LIN {X 0,Y 514.203,Z 355.204,A -85,B 0,C 180,E1 21211.136,E2 21211.136} C_VEL
LIN {X 0,Y 523.053,Z 367.857,A -85,B 0,C 180,E1 21208.99,E2 21208.99} C_VEL
LIN {X 0,Y 532.804,Z 382.486,A -85,B 0,C 180,E1 21206.835,E2 21206.835} C_VEL
LIN {X 0,Y 543.184,Z 399.298,A -85,B 0,C 180,E1 21204.725,E2 21204.725} C_VEL
LIN {X 0,Y 532.021,Z 628.307,A -85,B 0,C 180,E1 21201.248,E2 21201.248} C_VEL
LIN {X 0,Y 527.564,Z 720.114,A -85,B 0,C 180,E1 21199.84,E2 21199.84} C_VEL
LIN {X 0,Y 524.972,Z 748.17,A -85,B 0,C 180,E1 21199.261,E2 21199.261} C_VEL
LIN {X 0,Y 522.324,Z 769.234,A -85,B 0,C 180,E1 21198.682,E2 21198.682} C_VEL
LIN {X 0,Y 519.318,Z 789.292,A -85,B 0,C 180,E1 21198.004,E2 21198.004} C_VEL
LIN {X 0,Y 515.218,Z 813.189,A -85,B 0,C 180,E1 21197.024,E2 21197.024} C_VEL
LIN {X 0,Y 510.576,Z 836.113,A -85,B 0,C 180,E1 21195.868,E2 21195.868} C_VEL
LIN {X 0,Y 506.148,Z 856.028,A -85,B 0,C 180,E1 21194.69,E2 21194.69} C_VEL
LIN {X 0,Y 500.798,Z 878.497,A -85,B 0,C 180,E1 21193.144,E2 21193.144} C_VEL
LIN {X 0,Y 495.189,Z 899.857,A -85,B 0,C 180,E1 21191.398,E2 21191.398} C_VEL
LIN {X 0,Y 490.436,Z 917.27,A -85,B 0,C 180,E1 21189.77,E2 21189.77} C_VEL
LIN {X 0,Y 484.861,Z 937.229,A -85,B 0,C 180,E1 21187.637,E2 21187.637} C_VEL
LIN {X 0,Y 479.642,Z 955.131,A -85,B 0,C 180,E1 21185.402,E2 21185.402} C_VEL
LIN {X 0,Y 475.369,Z 969.999,A -85,B 0,C 180,E1 21183.297,E2 21183.297} C_VEL
LIN {X 0,Y 470.786,Z 986.437,A -85,B 0,C 180,E1 21180.646,E2 21180.646} C_VEL
LIN {X 0,Y 466.894,Z 1000.666,A -85,B 0,C 180,E1 21177.97,E2 21177.97} C_VEL
LIN {X 0,Y 463.87,Z 1012.654,A -85,B 0,C 180,E1 21175.401,E2 21175.401} C_VEL
LIN {X 0,Y 460.826,Z 1026.036,A -85,B 0,C 180,E1 21172.047,E2 21172.047} C_VEL
LIN {X 0,Y 459.016,Z 1035.196,A -85,B 0,C 180,E1 21169.336,E2 21169.336} C_VEL
LIN {X 0,Y 457.668,Z 1043.402,A -85,B 0,C 180,E1 21166.5,E2 21166.5} C_VEL
LIN {X 0,Y 456.674,Z 1051.232,A -85,B 0,C 180,E1 21163.162,E2 21163.162} C_VEL
LIN {X 0,Y 456.221,Z 1056.208,A -85,B 0,C 180,E1 21160.481,E2 21160.481} C_VEL
LIN {X 0,Y 456.026,Z 1059.887,A -85,B 0,C 180,E1 21157.94,E2 21157.94} C_VEL
LIN {X 0,Y 455.923,Z 1062.661,A -85,B 0,C 180,E1 21155.285,E2 21155.285} C_VEL
LIN {X 0,Y 455.906,Z 1064.554,A -85,B 0,C 180,E1 21152.137,E2 21152.137} C_VEL
LIN {X 0,Y 455.907,Z 1064.806,A -85,B 0,C 180,E1 21149.246,E2 21149.246} C_VEL
LIN {X 0,Y 455.911,Z 1063.998,A -85,B 0,C 180,E1 21146.731,E2 21146.731} C_VEL
LIN {X 0,Y 455.927,Z 1062.196,A -85,B 0,C 180,E1 21144.21,E2 21144.21} C_VEL
LIN {X 0,Y 456.039,Z 1059.388,A -85,B 0,C 180,E1 21141.68,E2 21141.68} C_VEL
LIN {X 0,Y 456.344,Z 1054.717,A -85,B 0,C 180,E1 21138.627,E2 21138.627} C_VEL
LIN {X 0,Y 457.032,Z 1048.041,A -85,B 0,C 180,E1 21135.428,E2 21135.428} C_VEL
LIN {X 0,Y 457.983,Z 1041.122,A -85,B 0,C 180,E1 21132.727,E2 21132.727} C_VEL
LIN {X 0,Y 459.607,Z 1031.801,A -85,B 0,C 180,E1 21129.662,E2 21129.662} C_VEL
LIN {X 0,Y 461.885,Z 1020.576,A -85,B 0,C 180,E1 21126.618,E2 21126.618} C_VEL
LIN {X 0,Y 464.343,Z 1009.773,A -85,B 0,C 180,E1 21124.079,E2 21124.079} C_VEL
LIN {X 0,Y 467.932,Z 995.579,A -85,B 0,C 180,E1 21121.176,E2 21121.176} C_VEL
LIN {X 0,Y 471.825,Z 980.703,A -85,B 0,C 180,E1 21118.579,E2 21118.579} C_VEL
LIN {X 0,Y 475.618,Z 966.792,A -85,B 0,C 180,E1 21116.434,E2 21116.434} C_VEL
LIN {X 0,Y 480.739,Z 948.351,A -85,B 0,C 180,E1 21113.942,E2 21113.942} C_VEL
LIN {X 0,Y 485.605,Z 930.371,A -85,B 0,C 180,E1 21111.851,E2 21111.851} C_VEL
LIN {X 0,Y 490.241,Z 913.03,A -85,B 0,C 180,E1 21110.075,E2 21110.075} C_VEL
LIN {X 0,Y 496.23,Z 889.626,A -85,B 0,C 180,E1 21108.013,E2 21108.013} C_VEL
LIN {X 0,Y 500.877,Z 870.253,A -85,B 0,C 180,E1 21106.551,E2 21106.551} C_VEL
LIN {X 0,Y 505.83,Z 848.283,A -85,B 0,C 180,E1 21105.115,E2 21105.115} C_VEL
LIN {X 0,Y 510.392,Z 825.521,A -85,B 0,C 180,E1 21103.869,E2 21103.869} C_VEL
LIN {X 0,Y 514.144,Z 804.539,A -85,B 0,C 180,E1 21102.896,E2 21102.896} C_VEL
LIN {X 0,Y 517.885,Z 780.938,A -85,B 0,C 180,E1 21101.985,E2 21101.985} C_VEL
LIN {X 0,Y 521.183,Z 755.093,A -85,B 0,C 180,E1 21101.206,E2 21101.206} C_VEL
LIN {X 0,Y 523.436,Z 733.002,A -85,B 0,C 180,E1 21100.696,E2 21100.696} C_VEL
LIN {X 0,Y 525.243,Z 706.485,A -85,B 0,C 180,E1 21100.229,E2 21100.229} C_VEL
LIN {X 0,Y 535.513,Z 472.628,A -85,B 0,C 180,E1 21096.713,E2 21096.713} C_VEL
LIN {X 0,Y 538.83,Z 397.459,A -85,B 0,C 180,E1 21095.558,E2 21095.558} C_VEL
LIN {X 0,Y 529.792,Z 382.604,A -85,B 0,C 180,E1 21093.897,E2 21093.897} C_VEL
LIN {X 0,Y 520.675,Z 368.292,A -85,B 0,C 180,E1 21092.105,E2 21092.105} C_VEL
LIN {X 0,Y 510.021,Z 352.551,A -85,B 0,C 180,E1 21089.833,E2 21089.833} C_VEL
LIN {X 0,Y 499.991,Z 338.758,A -85,B 0,C 180,E1 21087.481,E2 21087.481} C_VEL
LIN {X 0,Y 494.424,Z 331.393,A -85,B 0,C 180,E1 21086.063,E2 21086.063} C_VEL
LIN {X 0,Y 490.131,Z 326.165,A -85,B 0,C 180,E1 21084.915,E2 21084.915} C_VEL
LIN {X 0,Y 486.39,Z 321.608,A -85,B 0,C 180,E1 21083.858,E2 21083.858} C_VEL
LIN {X 0,Y 481.772,Z 316.366,A -85,B 0,C 180,E1 21082.483,E2 21082.483} C_VEL
LIN {X 0,Y 480.461,Z 314.61,A -85,B 0,C 180,E1 21082.064,E2 21082.064} C_VEL
LIN {X 0,Y 477.038,Z 311.21,A -85,B 0,C 180,E1 21080.971,E2 21080.971} C_VEL
LIN {X 0,Y 475.539,Z 308.65,A -85,B 0,C 180,E1 21080.429,E2 21080.429} C_VEL
LIN {X 0,Y 472.204,Z 306.004,A -85,B 0,C 180,E1 21079.289,E2 21079.289} C_VEL
LIN {X 0,Y 469.864,Z 302.242,A -85,B 0,C 180,E1 21078.358,E2 21078.358} C_VEL
LIN {X 0,Y 466.516,Z 299.897,A -85,B 0,C 180,E1 21077.076,E2 21077.076} C_VEL
LIN {X 0,Y 464.568,Z 296.605,A -85,B 0,C 180,E1 21076.184,E2 21076.184} C_VEL
LIN {X 0,Y 463.641,Z 295.554,A -85,B 0,C 180,E1 21075.767,E2 21075.767} C_VEL
LIN {X 0,Y 460.216,Z 293.29,A -85,B 0,C 180,E1 21074.212,E2 21074.212} C_VEL
LIN {X 0,Y 458.544,Z 290.48,A -85,B 0,C 180,E1 21073.268,E2 21073.268} C_VEL
LIN {X 0,Y 458.252,Z 289.079,A -85,B 0,C 180,E1 21072.603,E2 21072.603} C_VEL
LIN {X 0,Y 458.192,Z 288.875,A -85,B 0,C 180,E1 21068.913,E2 21068.913} C_VEL
LIN {X 0,Y 458.169,Z 288.888,A -85,B 0,C 180,E1 21065.385,E2 21065.385} C_VEL
LIN {X 0,Y 458.176,Z 288.901,A -85,B 0,C 180,E1 21061.626,E2 21061.626} C_VEL
LIN {X 0,Y 458.207,Z 288.898,A -85,B 0,C 180,E1 21058.066,E2 21058.066} C_VEL
LIN {X 0,Y 458.22,Z 288.88,A -85,B 0,C 180,E1 21054.365,E2 21054.365} C_VEL
LIN {X 0,Y 458.176,Z 288.875,A -85,B 0,C 180,E1 21050.833,E2 21050.833} C_VEL
LIN {X 0,Y 458.167,Z 288.876,A -85,B 0,C 180,E1 21047.266,E2 21047.266} C_VEL
LIN {X 0,Y 458.249,Z 289.067,A -85,B 0,C 180,E1 21044.172,E2 21044.172} C_VEL
LIN {X 0,Y 458.531,Z 290.412,A -85,B 0,C 180,E1 21043.564,E2 21043.564} C_VEL
LIN {X 0,Y 460.199,Z 293.267,A -85,B 0,C 180,E1 21042.617,E2 21042.617} C_VEL
LIN {X 0,Y 464.437,Z 296.312,A -85,B 0,C 180,E1 21040.703,E2 21040.703} C_VEL
LIN {X 0,Y 466.371,Z 299.715,A -85,B 0,C 180,E1 21039.807,E2 21039.807} C_VEL
LIN {X 0,Y 469.38,Z 302.008,A -85,B 0,C 180,E1 21038.637,E2 21038.637} C_VEL
LIN {X 0,Y 470.174,Z 302.632,A -85,B 0,C 180,E1 21038.341,E2 21038.341} C_VEL
LIN {X 0,Y 472.366,Z 306.213,A -85,B 0,C 180,E1 21037.472,E2 21037.472} C_VEL
LIN {X 0,Y 475.79,Z 309.044,A -85,B 0,C 180,E1 21036.302,E2 21036.302} C_VEL
LIN {X 0,Y 478.497,Z 312.895,A -85,B 0,C 180,E1 21035.366,E2 21035.366} C_VEL
LIN {X 0,Y 481.207,Z 315.37,A -85,B 0,C 180,E1 21034.525,E2 21034.525} C_VEL
LIN {X 0,Y 484.441,Z 319.575,A -85,B 0,C 180,E1 21033.524,E2 21033.524} C_VEL
LIN {X 0,Y 486.437,Z 321.649,A -85,B 0,C 180,E1 21032.949,E2 21032.949} C_VEL
LIN {X 0,Y 490.194,Z 326.225,A -85,B 0,C 180,E1 21031.888,E2 21031.888} C_VEL
LIN {X 0,Y 496.779,Z 334.239,A -85,B 0,C 180,E1 21030.155,E2 21030.155} C_VEL
LIN {X 0,Y 501.543,Z 340.256,A -85,B 0,C 180,E1 21028.979,E2 21028.979} C_VEL
LIN {X 0,Y 509.07,Z 349.89,A -85,B 0,C 180,E1 21027.24,E2 21027.24} C_VEL
LIN {X 0,Y 518.285,Z 362.361,A -85,B 0,C 180,E1 21025.27,E2 21025.27} C_VEL
LIN {X 0,Y 529.578,Z 379.496,A -85,B 0,C 180,E1 21023.033,E2 21023.033} C_VEL
LIN {X 0,Y 538.954,Z 394.907,A -85,B 0,C 180,E1 21021.302,E2 21021.302} C_VEL
LIN {X 0,Y 529.781,Z 598.454,A -85,B 0,C 180,E1 21018.226,E2 21018.226} C_VEL
LIN {X 0,Y 524.636,Z 713.049,A -85,B 0,C 180,E1 21016.486,E2 21016.486} C_VEL
LIN {X 0,Y 522.257,Z 740.771,A -85,B 0,C 180,E1 21015.915,E2 21015.915} C_VEL
LIN {X 0,Y 519.645,Z 763.002,A -85,B 0,C 180,E1 21015.295,E2 21015.295} C_VEL
LIN {X 0,Y 516.831,Z 782.979,A -85,B 0,C 180,E1 21014.61,E2 21014.61} C_VEL
LIN {X 0,Y 512.992,Z 806.654,A -85,B 0,C 180,E1 21013.629,E2 21013.629} C_VEL
LIN {X 0,Y 508.642,Z 829.268,A -85,B 0,C 180,E1 21012.481,E2 21012.481} C_VEL
LIN {X 0,Y 504.692,Z 847.952,A -85,B 0,C 180,E1 21011.378,E2 21011.378} C_VEL
LIN {X 0,Y 500.224,Z 867.614,A -85,B 0,C 180,E1 21010.042,E2 21010.042} C_VEL
LIN {X 0,Y 494.587,Z 890.568,A -85,B 0,C 180,E1 21008.216,E2 21008.216} C_VEL
LIN {X 0,Y 489.946,Z 908.319,A -85,B 0,C 180,E1 21006.578,E2 21006.578} C_VEL
LIN {X 0,Y 485.351,Z 925.361,A -85,B 0,C 180,E1 21004.796,E2 21004.796} C_VEL
LIN {X 0,Y 479.796,Z 945.368,A -85,B 0,C 180,E1 21002.383,E2 21002.383} C_VEL
LIN {X 0,Y 475.603,Z 960.328,A -85,B 0,C 180,E1 21000.302,E2 21000.302} C_VEL
LIN {X 0,Y 471.696,Z 974.528,A -85,B 0,C 180,E1 20998.072,E2 20998.072} C_VEL
LIN {X 0,Y 470.388,Z 979.442,A -85,B 0,C 180,E1 20997.234,E2 20997.234} C_VEL
LIN {X 0,Y 468.274,Z 983.858,A -85,B 0,C 180,E1 20996.497,E2 20996.497} C_VEL
LIN {X 0,Y 459.467,Z 995.612,A -85,B 0,C 180,E1 20994.601,E2 20994.601} C_VEL
LIN {X 0,Y 457.85,Z 998.982,A -85,B 0,C 180,E1 20993.913,E2 20993.913} C_VEL
LIN {X 0,Y 454.838,Z 1010.772,A -85,B 0,C 180,E1 20991.132,E2 20991.132} C_VEL
LIN {X 0,Y 452.659,Z 1020.323,A -85,B 0,C 180,E1 20988.547,E2 20988.547} C_VEL
LIN {X 0,Y 450.633,Z 1030.545,A -85,B 0,C 180,E1 20985.31,E2 20985.31} C_VEL
LIN {X 0,Y 449.378,Z 1038.199,A -85,B 0,C 180,E1 20982.334,E2 20982.334} C_VEL
LIN {X 0,Y 448.644,Z 1043.977,A -85,B 0,C 180,E1 20979.622,E2 20979.622} C_VEL
LIN {X 0,Y 448.188,Z 1049.021,A -85,B 0,C 180,E1 20976.662,E2 20976.662} C_VEL
LIN {X 0,Y 447.969,Z 1053.013,A -85,B 0,C 180,E1 20973.327,E2 20973.327} C_VEL
LIN {X 0,Y 447.928,Z 1055.023,A -85,B 0,C 180,E1 20970.639,E2 20970.639} C_VEL
LIN {X 0,Y 447.907,Z 1055.948,A -85,B 0,C 180,E1 20968.081,E2 20968.081} C_VEL
LIN {X 0,Y 447.905,Z 1055.901,A -85,B 0,C 180,E1 20965.519,E2 20965.519} C_VEL
LIN {X 0,Y 447.921,Z 1054.74,A -85,B 0,C 180,E1 20962.69,E2 20962.69} C_VEL
LIN {X 0,Y 448.033,Z 1051.756,A -85,B 0,C 180,E1 20959.325,E2 20959.325} C_VEL
LIN {X 0,Y 448.263,Z 1047.994,A -85,B 0,C 180,E1 20956.542,E2 20956.542} C_VEL
LIN {X 0,Y 448.757,Z 1043.183,A -85,B 0,C 180,E1 20953.808,E2 20953.808} C_VEL
LIN {X 0,Y 449.736,Z 1036.286,A -85,B 0,C 180,E1 20950.654,E2 20950.654} C_VEL
LIN {X 0,Y 451.296,Z 1027.48,A -85,B 0,C 180,E1 20947.462,E2 20947.462} C_VEL
LIN {X 0,Y 453.17,Z 1018.757,A -85,B 0,C 180,E1 20944.775,E2 20944.775} C_VEL
LIN {X 0,Y 456.012,Z 1007.309,A -85,B 0,C 180,E1 20941.731,E2 20941.731} C_VEL
LIN {X 0,Y 459.523,Z 994.09,A -85,B 0,C 180,E1 20938.776,E2 20938.776} C_VEL
LIN {X 0,Y 463.198,Z 981.437,A -85,B 0,C 180,E1 20936.305,E2 20936.305} C_VEL
LIN {X 0,Y 468.021,Z 965.359,A -85,B 0,C 180,E1 20933.564,E2 20933.564} C_VEL
LIN {X 0,Y 472.912,Z 949.158,A -85,B 0,C 180,E1 20931.194,E2 20931.194} C_VEL
LIN {X 0,Y 477.748,Z 933.313,A -85,B 0,C 180,E1 20929.153,E2 20929.153} C_VEL
LIN {X 0,Y 483.979,Z 912.441,A -85,B 0,C 180,E1 20926.827,E2 20926.827} C_VEL
LIN {X 0,Y 489.009,Z 894.83,A -85,B 0,C 180,E1 20925.136,E2 20925.136} C_VEL
LIN {X 0,Y 493.881,Z 877.04,A -85,B 0,C 180,E1 20923.633,E2 20923.633} C_VEL
LIN {X 0,Y 499.693,Z 854.414,A -85,B 0,C 180,E1 20921.981,E2 20921.981} C_VEL
LIN {X 0,Y 504.539,Z 833.5,A -85,B 0,C 180,E1 20920.693,E2 20920.693} C_VEL
LIN {X 0,Y 508.601,Z 814.32,A -85,B 0,C 180,E1 20919.676,E2 20919.676} C_VEL
LIN {X 0,Y 512.859,Z 791.904,A -85,B 0,C 180,E1 20918.664,E2 20918.664} C_VEL
LIN {X 0,Y 516.841,Z 766.821,A -85,B 0,C 180,E1 20917.754,E2 20917.754} C_VEL
LIN {X 0,Y 519.62,Z 745.455,A -85,B 0,C 180,E1 20917.132,E2 20917.132} C_VEL
LIN {X 0,Y 522.147,Z 721.367,A -85,B 0,C 180,E1 20916.592,E2 20916.592} C_VEL
LIN {X 0,Y 524.302,Z 685.323,A -85,B 0,C 180,E1 20916.003,E2 20916.003} C_VEL
LIN {X 0,Y 535.535,Z 458.38,A -85,B 0,C 180,E1 20912.543,E2 20912.543} C_VEL
LIN {X 0,Y 538.44,Z 400.484,A -85,B 0,C 180,E1 20911.642,E2 20911.642} C_VEL
LIN {X 0,Y 529.82,Z 386.785,A -85,B 0,C 180,E1 20909.852,E2 20909.852} C_VEL
LIN {X 0,Y 520.026,Z 372.01,A -85,B 0,C 180,E1 20907.637,E2 20907.637} C_VEL
LIN {X 0,Y 512.262,Z 361.699,A -85,B 0,C 180,E1 20905.741,E2 20905.741} C_VEL
LIN {X 0,Y 504.417,Z 351.549,A -85,B 0,C 180,E1 20903.635,E2 20903.635} C_VEL
LIN {X 0,Y 499.945,Z 346.055,A -85,B 0,C 180,E1 20902.334,E2 20902.334} C_VEL
LIN {X 0,Y 495.787,Z 340.957,A -85,B 0,C 180,E1 20901.038,E2 20901.038} C_VEL
LIN {X 0,Y 491.944,Z 336.155,A -85,B 0,C 180,E1 20899.75,E2 20899.75} C_VEL
LIN {X 0,Y 487.525,Z 331.174,A -85,B 0,C 180,E1 20898.165,E2 20898.165} C_VEL
LIN {X 0,Y 486.227,Z 329.433,A -85,B 0,C 180,E1 20897.657,E2 20897.657} C_VEL
LIN {X 0,Y 482.681,Z 325.856,A -85,B 0,C 180,E1 20896.24,E2 20896.24} C_VEL
LIN {X 0,Y 480.9,Z 323.244,A -85,B 0,C 180,E1 20895.435,E2 20895.435} C_VEL
LIN {X 0,Y 477.612,Z 320.364,A -85,B 0,C 180,E1 20893.931,E2 20893.931} C_VEL
LIN {X 0,Y 475.685,Z 317.08,A -85,B 0,C 180,E1 20892.874,E2 20892.874} C_VEL
LIN {X 0,Y 471.969,Z 314.314,A -85,B 0,C 180,E1 20890.807,E2 20890.807} C_VEL
LIN {X 0,Y 470.14,Z 311.069,A -85,B 0,C 180,E1 20889.487,E2 20889.487} C_VEL
LIN {X 0,Y 468.4,Z 309.861,A -85,B 0,C 180,E1 20888.223,E2 20888.223} C_VEL
LIN {X 0,Y 465.191,Z 306.945,A -85,B 0,C 180,E1 20885.18,E2 20885.18} C_VEL
LIN {X 0,Y 463.918,Z 304.394,A -85,B 0,C 180,E1 20883.212,E2 20883.212} C_VEL
LIN {X 0,Y 462.586,Z 303.371,A -85,B 0,C 180,E1 20879.628,E2 20879.628} C_VEL
LIN {X 0,Y 463.555,Z 304.007,A -85,B 0,C 180,E1 20874.554,E2 20874.554} C_VEL
LIN {X 0,Y 464.244,Z 304.979,A -85,B 0,C 180,E1 20873.321,E2 20873.321} C_VEL
LIN {X 0,Y 466.922,Z 308.959,A -85,B 0,C 180,E1 20870.084,E2 20870.084} C_VEL
LIN {X 0,Y 470.086,Z 310.878,A -85,B 0,C 180,E1 20867.657,E2 20867.657} C_VEL
LIN {X 0,Y 472,Z 314.284,A -85,B 0,C 180,E1 20866.275,E2 20866.275} C_VEL
LIN {X 0,Y 475.363,Z 316.917,A -85,B 0,C 180,E1 20864.381,E2 20864.381} C_VEL
LIN {X 0,Y 476.013,Z 317.736,A -85,B 0,C 180,E1 20864.028,E2 20864.028} C_VEL
LIN {X 0,Y 478.473,Z 321.384,A -85,B 0,C 180,E1 20862.738,E2 20862.738} C_VEL
LIN {X 0,Y 481.532,Z 323.91,A -85,B 0,C 180,E1 20861.382,E2 20861.382} C_VEL
LIN {X 0,Y 484.662,Z 328.131,A -85,B 0,C 180,E1 20860.035,E2 20860.035} C_VEL
LIN {X 0,Y 486.875,Z 330.162,A -85,B 0,C 180,E1 20859.189,E2 20859.189} C_VEL
LIN {X 0,Y 490.157,Z 334.487,A -85,B 0,C 180,E1 20857.954,E2 20857.954} C_VEL
LIN {X 0,Y 492.165,Z 336.566,A -85,B 0,C 180,E1 20857.262,E2 20857.262} C_VEL
LIN {X 0,Y 496.052,Z 341.208,A -85,B 0,C 180,E1 20855.973,E2 20855.973} C_VEL
LIN {X 0,Y 503.837,Z 351.484,A -85,B 0,C 180,E1 20853.606,E2 20853.606} C_VEL
LIN {X 0,Y 511.816,Z 362.382,A -85,B 0,C 180,E1 20851.435,E2 20851.435} C_VEL
LIN {X 0,Y 520.244,Z 374.603,A -85,B 0,C 180,E1 20849.349,E2 20849.349} C_VEL
LIN {X 0,Y 529.986,Z 389.406,A -85,B 0,C 180,E1 20847.152,E2 20847.152} C_VEL
LIN {X 0,Y 538.508,Z 403.514,A -85,B 0,C 180,E1 20845.37,E2 20845.37} C_VEL
LIN {X 0,Y 526.986,Z 632.03,A -85,B 0,C 180,E1 20841.883,E2 20841.883} C_VEL
LIN {X 0,Y 522.548,Z 720.163,A -85,B 0,C 180,E1 20840.523,E2 20840.523} C_VEL
LIN {X 0,Y 519.868,Z 748.294,A -85,B 0,C 180,E1 20839.94,E2 20839.94} C_VEL
LIN {X 0,Y 517.168,Z 769.128,A -85,B 0,C 180,E1 20839.366,E2 20839.366} C_VEL
LIN {X 0,Y 513.985,Z 789.723,A -85,B 0,C 180,E1 20838.669,E2 20838.669} C_VEL
LIN {X 0,Y 509.53,Z 814.676,A -85,B 0,C 180,E1 20837.632,E2 20837.632} C_VEL
LIN {X 0,Y 504.755,Z 837.376,A -85,B 0,C 180,E1 20836.471,E2 20836.471} C_VEL
LIN {X 0,Y 500.151,Z 857.345,A -85,B 0,C 180,E1 20835.274,E2 20835.274} C_VEL
LIN {X 0,Y 494.381,Z 880.483,A -85,B 0,C 180,E1 20833.648,E2 20833.648} C_VEL
LIN {X 0,Y 489.062,Z 900,A -85,B 0,C 180,E1 20832.034,E2 20832.034} C_VEL
LIN {X 0,Y 484.209,Z 917.111,A -85,B 0,C 180,E1 20830.421,E2 20830.421} C_VEL
LIN {X 0,Y 478.43,Z 937.028,A -85,B 0,C 180,E1 20828.276,E2 20828.276} C_VEL
LIN {X 0,Y 472.943,Z 955.1,A -85,B 0,C 180,E1 20825.997,E2 20825.997} C_VEL
LIN {X 0,Y 468.449,Z 970.051,A -85,B 0,C 180,E1 20823.855,E2 20823.855} C_VEL
LIN {X 0,Y 463.488,Z 986.963,A -85,B 0,C 180,E1 20821.079,E2 20821.079} C_VEL
LIN {X 0,Y 459.565,Z 1000.679,A -85,B 0,C 180,E1 20818.456,E2 20818.456} C_VEL
LIN {X 0,Y 456.368,Z 1012.654,A -85,B 0,C 180,E1 20815.849,E2 20815.849} C_VEL
LIN {X 0,Y 453.258,Z 1025.557,A -85,B 0,C 180,E1 20812.572,E2 20812.572} C_VEL
LIN {X 0,Y 451.312,Z 1034.761,A -85,B 0,C 180,E1 20809.814,E2 20809.814} C_VEL
LIN {X 0,Y 449.91,Z 1042.655,A -85,B 0,C 180,E1 20807.059,E2 20807.059} C_VEL
LIN {X 0,Y 448.796,Z 1050.668,A -85,B 0,C 180,E1 20803.66,E2 20803.66} C_VEL
LIN {X 0,Y 448.271,Z 1055.941,A -85,B 0,C 180,E1 20800.799,E2 20800.799} C_VEL
LIN {X 0,Y 448.036,Z 1059.661,A -85,B 0,C 180,E1 20798.212,E2 20798.212} C_VEL
LIN {X 0,Y 447.924,Z 1062.363,A -85,B 0,C 180,E1 20795.637,E2 20795.637} C_VEL
LIN {X 0,Y 447.913,Z 1064.271,A -85,B 0,C 180,E1 20792.687,E2 20792.687} C_VEL
LIN {X 0,Y 447.903,Z 1064.771,A -85,B 0,C 180,E1 20789.488,E2 20789.488} C_VEL
LIN {X 0,Y 447.912,Z 1063.984,A -85,B 0,C 180,E1 20786.801,E2 20786.801} C_VEL
LIN {X 0,Y 447.932,Z 1062.109,A -85,B 0,C 180,E1 20784.106,E2 20784.106} C_VEL
LIN {X 0,Y 448.048,Z 1059.295,A -85,B 0,C 180,E1 20781.53,E2 20781.53} C_VEL
LIN {X 0,Y 448.378,Z 1054.618,A -85,B 0,C 180,E1 20778.422,E2 20778.422} C_VEL
LIN {X 0,Y 449.108,Z 1047.928,A -85,B 0,C 180,E1 20775.165,E2 20775.165} C_VEL
LIN {X 0,Y 450.068,Z 1041.357,A -85,B 0,C 180,E1 20772.547,E2 20772.547} C_VEL
LIN {X 0,Y 451.615,Z 1032.797,A -85,B 0,C 180,E1 20769.659,E2 20769.659} C_VEL
LIN {X 0,Y 454.14,Z 1020.96,A -85,B 0,C 180,E1 20766.337,E2 20766.337} C_VEL
LIN {X 0,Y 456.71,Z 1010.19,A -85,B 0,C 180,E1 20763.753,E2 20763.753} C_VEL
LIN {X 0,Y 460.33,Z 996.509,A -85,B 0,C 180,E1 20760.886,E2 20760.886} C_VEL
LIN {X 0,Y 464.495,Z 981.283,A -85,B 0,C 180,E1 20758.171,E2 20758.171} C_VEL
LIN {X 0,Y 468.431,Z 967.433,A -85,B 0,C 180,E1 20755.996,E2 20755.996} C_VEL
LIN {X 0,Y 473.547,Z 949.831,A -85,B 0,C 180,E1 20753.56,E2 20753.56} C_VEL
LIN {X 0,Y 478.768,Z 931.23,A -85,B 0,C 180,E1 20751.358,E2 20751.358} C_VEL
LIN {X 0,Y 483.517,Z 914.117,A -85,B 0,C 180,E1 20749.579,E2 20749.579} C_VEL
LIN {X 0,Y 489.181,Z 893.05,A -85,B 0,C 180,E1 20747.667,E2 20747.667} C_VEL
LIN {X 0,Y 494.367,Z 872.191,A -85,B 0,C 180,E1 20746.058,E2 20746.058} C_VEL
LIN {X 0,Y 498.973,Z 852.442,A -85,B 0,C 180,E1 20744.734,E2 20744.734} C_VEL
LIN {X 0,Y 504.099,Z 828.48,A -85,B 0,C 180,E1 20743.368,E2 20743.368} C_VEL
LIN {X 0,Y 508.303,Z 805.834,A -85,B 0,C 180,E1 20742.3,E2 20742.3} C_VEL
LIN {X 0,Y 511.842,Z 784.287,A -85,B 0,C 180,E1 20741.451,E2 20741.451} C_VEL
LIN {X 0,Y 515.633,Z 756.398,A -85,B 0,C 180,E1 20740.582,E2 20740.582} C_VEL
LIN {X 0,Y 518.022,Z 733.825,A -85,B 0,C 180,E1 20740.054,E2 20740.054} C_VEL
LIN {X 0,Y 519.83,Z 708.889,A -85,B 0,C 180,E1 20739.606,E2 20739.606} C_VEL
LIN {X 0,Y 530.5,Z 474.753,A -85,B 0,C 180,E1 20736.063,E2 20736.063} C_VEL
LIN {X 0,Y 533.891,Z 401.34,A -85,B 0,C 180,E1 20734.933,E2 20734.933} C_VEL
LIN {X 0,Y 521.929,Z 381.65,A -85,B 0,C 180,E1 20732.635,E2 20732.635} C_VEL
LIN {X 0,Y 508.905,Z 361.823,A -85,B 0,C 180,E1 20729.873,E2 20729.873} C_VEL
LIN {X 0,Y 498.161,Z 346.708,A -85,B 0,C 180,E1 20727.332,E2 20727.332} C_VEL
LIN {X 0,Y 491.924,Z 338.422,A -85,B 0,C 180,E1 20725.719,E2 20725.719} C_VEL
LIN {X 0,Y 487.786,Z 333.333,A -85,B 0,C 180,E1 20724.59,E2 20724.59} C_VEL
LIN {X 0,Y 483.919,Z 328.472,A -85,B 0,C 180,E1 20723.47,E2 20723.47} C_VEL
LIN {X 0,Y 479.72,Z 323.762,A -85,B 0,C 180,E1 20722.197,E2 20722.197} C_VEL
LIN {X 0,Y 478.423,Z 322.035,A -85,B 0,C 180,E1 20721.776,E2 20721.776} C_VEL
LIN {X 0,Y 474.893,Z 318.339,A -85,B 0,C 180,E1 20720.619,E2 20720.619} C_VEL
LIN {X 0,Y 473.389,Z 316.057,A -85,B 0,C 180,E1 20720.074,E2 20720.074} C_VEL
LIN {X 0,Y 469.99,Z 312.974,A -85,B 0,C 180,E1 20718.867,E2 20718.867} C_VEL
LIN {X 0,Y 467.967,Z 309.826,A -85,B 0,C 180,E1 20718.048,E2 20718.048} C_VEL
LIN {X 0,Y 464.701,Z 307.27,A -85,B 0,C 180,E1 20716.758,E2 20716.758} C_VEL
LIN {X 0,Y 462.413,Z 303.43,A -85,B 0,C 180,E1 20715.682,E2 20715.682} C_VEL
LIN {X 0,Y 458.881,Z 301.098,A -85,B 0,C 180,E1 20714.061,E2 20714.061} C_VEL
LIN {X 0,Y 456.968,Z 298.081,A -85,B 0,C 180,E1 20712.993,E2 20712.993} C_VEL
LIN {X 0,Y 455.974,Z 296.632,A -85,B 0,C 180,E1 20712.41,E2 20712.41} C_VEL
LIN {X 0,Y 452.444,Z 294.447,A -85,B 0,C 180,E1 20710.312,E2 20710.312} C_VEL
LIN {X 0,Y 450.678,Z 291.624,A -85,B 0,C 180,E1 20708.935,E2 20708.935} C_VEL
LIN {X 0,Y 450.328,Z 290.302,A -85,B 0,C 180,E1 20708.17,E2 20708.17} C_VEL
LIN {X 0,Y 450.253,Z 289.888,A -85,B 0,C 180,E1 20705.991,E2 20705.991} C_VEL
LIN {X 0,Y 450.28,Z 289.886,A -85,B 0,C 180,E1 20702.291,E2 20702.291} C_VEL
LIN {X 0,Y 450.254,Z 289.871,A -85,B 0,C 180,E1 20698.727,E2 20698.727} C_VEL
LIN {X 0,Y 450.229,Z 289.864,A -85,B 0,C 180,E1 20695.159,E2 20695.159} C_VEL
LIN {X 0,Y 450.233,Z 289.862,A -85,B 0,C 180,E1 20691.443,E2 20691.443} C_VEL
LIN {X 0,Y 450.298,Z 290.231,A -85,B 0,C 180,E1 20688.732,E2 20688.732} C_VEL
LIN {X 0,Y 450.691,Z 291.628,A -85,B 0,C 180,E1 20687.873,E2 20687.873} C_VEL
LIN {X 0,Y 452.34,Z 294.335,A -85,B 0,C 180,E1 20686.579,E2 20686.579} C_VEL
LIN {X 0,Y 455.62,Z 296.496,A -85,B 0,C 180,E1 20684.601,E2 20684.601} C_VEL
LIN {X 0,Y 456.723,Z 297.434,A -85,B 0,C 180,E1 20683.987,E2 20683.987} C_VEL
LIN {X 0,Y 458.522,Z 300.695,A -85,B 0,C 180,E1 20682.944,E2 20682.944} C_VEL
LIN {X 0,Y 461.991,Z 303.267,A -85,B 0,C 180,E1 20681.318,E2 20681.318} C_VEL
LIN {X 0,Y 462.731,Z 303.898,A -85,B 0,C 180,E1 20680.989,E2 20680.989} C_VEL
LIN {X 0,Y 464.988,Z 307.585,A -85,B 0,C 180,E1 20679.941,E2 20679.941} C_VEL
LIN {X 0,Y 468.353,Z 310.253,A -85,B 0,C 180,E1 20678.621,E2 20678.621} C_VEL
LIN {X 0,Y 470.937,Z 314.109,A -85,B 0,C 180,E1 20677.597,E2 20677.597} C_VEL
LIN {X 0,Y 473.908,Z 316.66,A -85,B 0,C 180,E1 20676.565,E2 20676.565} C_VEL
LIN {X 0,Y 477.043,Z 320.806,A -85,B 0,C 180,E1 20675.48,E2 20675.48} C_VEL
LIN {X 0,Y 479.175,Z 322.836,A -85,B 0,C 180,E1 20674.806,E2 20674.806} C_VEL
LIN {X 0,Y 482.755,Z 327.307,A -85,B 0,C 180,E1 20673.689,E2 20673.689} C_VEL
LIN {X 0,Y 484.432,Z 329.252,A -85,B 0,C 180,E1 20673.192,E2 20673.192} C_VEL
LIN {X 0,Y 488.468,Z 333.963,A -85,B 0,C 180,E1 20672.046,E2 20672.046} C_VEL
LIN {X 0,Y 493.057,Z 339.594,A -85,B 0,C 180,E1 20670.809,E2 20670.809} C_VEL
LIN {X 0,Y 502.322,Z 351.582,A -85,B 0,C 180,E1 20668.499,E2 20668.499} C_VEL
LIN {X 0,Y 513.061,Z 365.837,A -85,B 0,C 180,E1 20666.092,E2 20666.092} C_VEL
LIN {X 0,Y 523.157,Z 381.093,A -85,B 0,C 180,E1 20664.005,E2 20664.005} C_VEL
LIN {X 0,Y 533.472,Z 397.827,A -85,B 0,C 180,E1 20662.03,E2 20662.03} C_VEL
LIN {X 0,Y 533.979,Z 399.099,A -85,B 0,C 180,E1 20661.927,E2 20661.927} C_VEL
LIN {X 0,Y 524.465,Z 602.973,A -85,B 0,C 180,E1 20658.83,E2 20658.83} C_VEL
LIN {X 0,Y 519.337,Z 713.151,A -85,B 0,C 180,E1 20657.146,E2 20657.146} C_VEL
LIN {X 0,Y 516.893,Z 740.867,A -85,B 0,C 180,E1 20656.573,E2 20656.573} C_VEL
LIN {X 0,Y 514.218,Z 762.993,A -85,B 0,C 180,E1 20655.954,E2 20655.954} C_VEL
LIN {X 0,Y 511.414,Z 782.349,A -85,B 0,C 180,E1 20655.291,E2 20655.291} C_VEL
LIN {X 0,Y 507.471,Z 806.004,A -85,B 0,C 180,E1 20654.313,E2 20654.313} C_VEL
LIN {X 0,Y 502.924,Z 829.077,A -85,B 0,C 180,E1 20653.142,E2 20653.142} C_VEL
LIN {X 0,Y 498.65,Z 848.662,A -85,B 0,C 180,E1 20651.978,E2 20651.978} C_VEL
LIN {X 0,Y 493.58,Z 870.279,A -85,B 0,C 180,E1 20650.486,E2 20650.486} C_VEL
LIN {X 0,Y 488.136,Z 891.418,A -85,B 0,C 180,E1 20648.767,E2 20648.767} C_VEL
LIN {X 0,Y 483.448,Z 908.724,A -85,B 0,C 180,E1 20647.151,E2 20647.151} C_VEL
LIN {X 0,Y 478.583,Z 926.121,A -85,B 0,C 180,E1 20645.31,E2 20645.31} C_VEL
LIN {X 0,Y 472.928,Z 945.702,A -85,B 0,C 180,E1 20642.913,E2 20642.913} C_VEL
LIN {X 0,Y 468.562,Z 960.643,A -85,B 0,C 180,E1 20640.807,E2 20640.807} C_VEL
LIN {X 0,Y 464.28,Z 975.584,A -85,B 0,C 180,E1 20638.421,E2 20638.421} C_VEL
LIN {X 0,Y 459.872,Z 991.333,A -85,B 0,C 180,E1 20635.5,E2 20635.5} C_VEL
LIN {X 0,Y 457.85,Z 998.982,A -85,B 0,C 180,E1 20633.913,E2 20633.913} C_VEL
LIN {X 0,Y 455.895,Z 1002.818,A -85,B 0,C 180,E1 20633.101,E2 20633.101} C_VEL
LIN {X 0,Y 447.497,Z 1012.989,A -85,B 0,C 180,E1 20630.986,E2 20630.986} C_VEL
LIN {X 0,Y 446.056,Z 1015.869,A -85,B 0,C 180,E1 20630.239,E2 20630.239} C_VEL
LIN {X 0,Y 443.718,Z 1026.053,A -85,B 0,C 180,E1 20627.164,E2 20627.164} C_VEL
LIN {X 0,Y 442.211,Z 1033.862,A -85,B 0,C 180,E1 20624.402,E2 20624.402} C_VEL
LIN {X 0,Y 441.027,Z 1041.626,A -85,B 0,C 180,E1 20621.111,E2 20621.111} C_VEL
LIN {X 0,Y 440.363,Z 1047.328,A -85,B 0,C 180,E1 20617.961,E2 20617.961} C_VEL
LIN {X 0,Y 440.068,Z 1051.165,A -85,B 0,C 180,E1 20615.214,E2 20615.214} C_VEL
LIN {X 0,Y 439.938,Z 1053.915,A -85,B 0,C 180,E1 20612.475,E2 20612.475} C_VEL
LIN {X 0,Y 439.912,Z 1055.831,A -85,B 0,C 180,E1 20609.219,E2 20609.219} C_VEL
LIN {X 0,Y 439.902,Z 1056.084,A -85,B 0,C 180,E1 20606.09,E2 20606.09} C_VEL
LIN {X 0,Y 439.92,Z 1055.269,A -85,B 0,C 180,E1 20603.475,E2 20603.475} C_VEL
LIN {X 0,Y 439.96,Z 1053.47,A -85,B 0,C 180,E1 20600.846,E2 20600.846} C_VEL
LIN {X 0,Y 440.1,Z 1050.668,A -85,B 0,C 180,E1 20598.201,E2 20598.201} C_VEL
LIN {X 0,Y 440.554,Z 1045.769,A -85,B 0,C 180,E1 20594.87,E2 20594.87} C_VEL
LIN {X 0,Y 441.383,Z 1039.334,A -85,B 0,C 180,E1 20591.657,E2 20591.657} C_VEL
LIN {X 0,Y 442.511,Z 1032.736,A -85,B 0,C 180,E1 20588.941,E2 20588.941} C_VEL
LIN {X 0,Y 444.506,Z 1023.367,A -85,B 0,C 180,E1 20585.692,E2 20585.692} C_VEL
LIN {X 0,Y 447.155,Z 1012.42,A -85,B 0,C 180,E1 20582.572,E2 20582.572} C_VEL
LIN {X 0,Y 449.99,Z 1002.041,A -85,B 0,C 180,E1 20580.003,E2 20580.003} C_VEL
LIN {X 0,Y 454.062,Z 988.309,A -85,B 0,C 180,E1 20577.035,E2 20577.035} C_VEL
LIN {X 0,Y 458.721,Z 973.111,A -85,B 0,C 180,E1 20574.256,E2 20574.256} C_VEL
LIN {X 0,Y 463.195,Z 959.012,A -85,B 0,C 180,E1 20571.992,E2 20571.992} C_VEL
LIN {X 0,Y 469.008,Z 940.795,A -85,B 0,C 180,E1 20569.441,E2 20569.441} C_VEL
LIN {X 0,Y 474.401,Z 923.468,A -85,B 0,C 180,E1 20567.357,E2 20567.357} C_VEL
LIN {X 0,Y 479.653,Z 906.259,A -85,B 0,C 180,E1 20565.539,E2 20565.539} C_VEL
LIN {X 0,Y 486.112,Z 884.161,A -85,B 0,C 180,E1 20563.526,E2 20563.526} C_VEL
LIN {X 0,Y 491.326,Z 864.917,A -85,B 0,C 180,E1 20562.029,E2 20562.029} C_VEL
LIN {X 0,Y 496.383,Z 844.904,A -85,B 0,C 180,E1 20560.677,E2 20560.677} C_VEL
LIN {X 0,Y 502.19,Z 819.535,A -85,B 0,C 180,E1 20559.239,E2 20559.239} C_VEL
LIN {X 0,Y 506.263,Z 799.124,A -85,B 0,C 180,E1 20558.272,E2 20558.272} C_VEL
LIN {X 0,Y 510.03,Z 777.802,A -85,B 0,C 180,E1 20557.427,E2 20557.427} C_VEL
LIN {X 0,Y 514.027,Z 750.288,A -85,B 0,C 180,E1 20556.559,E2 20556.559} C_VEL
LIN {X 0,Y 516.592,Z 727.601,A -85,B 0,C 180,E1 20556.022,E2 20556.022} C_VEL
LIN {X 0,Y 518.508,Z 703.274,A -85,B 0,C 180,E1 20555.581,E2 20555.581} C_VEL
LIN {X 0,Y 530.49,Z 469.255,A -85,B 0,C 180,E1 20551.996,E2 20551.996} C_VEL
LIN {X 0,Y 533.792,Z 404.506,A -85,B 0,C 180,E1 20550.975,E2 20550.975} C_VEL
LIN {X 0,Y 524.258,Z 389.353,A -85,B 0,C 180,E1 20548.914,E2 20548.914} C_VEL
LIN {X 0,Y 516.074,Z 377.179,A -85,B 0,C 180,E1 20546.992,E2 20546.992} C_VEL
LIN {X 0,Y 509.473,Z 368.327,A -85,B 0,C 180,E1 20545.331,E2 20545.331} C_VEL
LIN {X 0,Y 502.035,Z 358.586,A -85,B 0,C 180,E1 20543.288,E2 20543.288} C_VEL
LIN {X 0,Y 497.721,Z 353.216,A -85,B 0,C 180,E1 20542.004,E2 20542.004} C_VEL
LIN {X 0,Y 493.794,Z 348.328,A -85,B 0,C 180,E1 20540.754,E2 20540.754} C_VEL
LIN {X 0,Y 489.856,Z 343.284,A -85,B 0,C 180,E1 20539.403,E2 20539.403} C_VEL
LIN {X 0,Y 485.801,Z 338.743,A -85,B 0,C 180,E1 20537.921,E2 20537.921} C_VEL
LIN {X 0,Y 484.521,Z 337.013,A -85,B 0,C 180,E1 20537.412,E2 20537.412} C_VEL
LIN {X 0,Y 480.905,Z 333.21,A -85,B 0,C 180,E1 20535.929,E2 20535.929} C_VEL
LIN {X 0,Y 479.406,Z 330.959,A -85,B 0,C 180,E1 20535.236,E2 20535.236} C_VEL
LIN {X 0,Y 476.052,Z 327.9,A -85,B 0,C 180,E1 20533.668,E2 20533.668} C_VEL
LIN {X 0,Y 474.26,Z 324.844,A -85,B 0,C 180,E1 20532.666,E2 20532.666} C_VEL
LIN {X 0,Y 470.527,Z 321.89,A -85,B 0,C 180,E1 20530.53,E2 20530.53} C_VEL
LIN {X 0,Y 468.593,Z 318.429,A -85,B 0,C 180,E1 20529.085,E2 20529.085} C_VEL
LIN {X 0,Y 464.516,Z 315.388,A -85,B 0,C 180,E1 20525.559,E2 20525.559} C_VEL
LIN {X 0,Y 462.801,Z 312.206,A -85,B 0,C 180,E1 20522.972,E2 20522.972} C_VEL
LIN {X 0,Y 461.563,Z 311.314,A -85,B 0,C 180,E1 20519.255,E2 20519.255} C_VEL
LIN {X 0,Y 462.646,Z 312.017,A -85,B 0,C 180,E1 20514.419,E2 20514.419} C_VEL
LIN {X 0,Y 463.257,Z 313.073,A -85,B 0,C 180,E1 20513.307,E2 20513.307} C_VEL
LIN {X 0,Y 465.899,Z 316.904,A -85,B 0,C 180,E1 20510.114,E2 20510.114} C_VEL
LIN {X 0,Y 468.78,Z 318.624,A -85,B 0,C 180,E1 20507.872,E2 20507.872} C_VEL
LIN {X 0,Y 470.749,Z 322.091,A -85,B 0,C 180,E1 20506.426,E2 20506.426} C_VEL
LIN {X 0,Y 474.443,Z 325.215,A -85,B 0,C 180,E1 20504.319,E2 20504.319} C_VEL
LIN {X 0,Y 477.026,Z 329.078,A -85,B 0,C 180,E1 20502.935,E2 20502.935} C_VEL
LIN {X 0,Y 479.97,Z 331.623,A -85,B 0,C 180,E1 20501.602,E2 20501.602} C_VEL
LIN {X 0,Y 483.28,Z 335.963,A -85,B 0,C 180,E1 20500.165,E2 20500.165} C_VEL
LIN {X 0,Y 485.239,Z 337.908,A -85,B 0,C 180,E1 20499.399,E2 20499.399} C_VEL
LIN {X 0,Y 488.734,Z 342.339,A -85,B 0,C 180,E1 20498.076,E2 20498.076} C_VEL
LIN {X 0,Y 490.393,Z 344.196,A -85,B 0,C 180,E1 20497.492,E2 20497.492} C_VEL
LIN {X 0,Y 495.406,Z 350.418,A -85,B 0,C 180,E1 20495.813,E2 20495.813} C_VEL
LIN {X 0,Y 501.659,Z 358.782,A -85,B 0,C 180,E1 20493.897,E2 20493.897} C_VEL
LIN {X 0,Y 509.443,Z 369.556,A -85,B 0,C 180,E1 20491.738,E2 20491.738} C_VEL
LIN {X 0,Y 517.559,Z 381.514,A -85,B 0,C 180,E1 20489.687,E2 20489.687} C_VEL
LIN {X 0,Y 527.073,Z 396.154,A -85,B 0,C 180,E1 20487.497,E2 20487.497} C_VEL
LIN {X 0,Y 533.905,Z 407.676,A -85,B 0,C 180,E1 20486.026,E2 20486.026} C_VEL
LIN {X 0,Y 522.054,Z 635.012,A -85,B 0,C 180,E1 20482.542,E2 20482.542} C_VEL
LIN {X 0,Y 517.612,Z 720.189,A -85,B 0,C 180,E1 20481.219,E2 20481.219} C_VEL
LIN {X 0,Y 514.856,Z 748.3,A -85,B 0,C 180,E1 20480.635,E2 20480.635} C_VEL
LIN {X 0,Y 512.067,Z 769.186,A -85,B 0,C 180,E1 20480.06,E2 20480.06} C_VEL
LIN {X 0,Y 508.726,Z 790.162,A -85,B 0,C 180,E1 20479.347,E2 20479.347} C_VEL
LIN {X 0,Y 504.134,Z 814.991,A -85,B 0,C 180,E1 20478.309,E2 20478.309} C_VEL
LIN {X 0,Y 499.217,Z 837.645,A -85,B 0,C 180,E1 20477.144,E2 20477.144} C_VEL
LIN {X 0,Y 494.577,Z 857.135,A -85,B 0,C 180,E1 20475.971,E2 20475.971} C_VEL
LIN {X 0,Y 488.597,Z 880.327,A -85,B 0,C 180,E1 20474.336,E2 20474.336} C_VEL
LIN {X 0,Y 483.079,Z 899.875,A -85,B 0,C 180,E1 20472.71,E2 20472.71} C_VEL
LIN {X 0,Y 477.97,Z 917.237,A -85,B 0,C 180,E1 20471.062,E2 20471.062} C_VEL
LIN {X 0,Y 471.999,Z 937.016,A -85,B 0,C 180,E1 20468.911,E2 20468.911} C_VEL
LIN {X 0,Y 466.265,Z 955.172,A -85,B 0,C 180,E1 20466.595,E2 20466.595} C_VEL
LIN {X 0,Y 461.576,Z 970.107,A -85,B 0,C 180,E1 20464.429,E2 20464.429} C_VEL
LIN {X 0,Y 456.31,Z 987.192,A -85,B 0,C 180,E1 20461.581,E2 20461.581} C_VEL
LIN {X 0,Y 452.269,Z 1000.695,A -85,B 0,C 180,E1 20458.958,E2 20458.958} C_VEL
LIN {X 0,Y 448.896,Z 1012.659,A -85,B 0,C 180,E1 20456.312,E2 20456.312} C_VEL
LIN {X 0,Y 445.614,Z 1025.542,A -85,B 0,C 180,E1 20452.981,E2 20452.981} C_VEL
LIN {X 0,Y 443.551,Z 1034.735,A -85,B 0,C 180,E1 20450.176,E2 20450.176} C_VEL
LIN {X 0,Y 442.046,Z 1042.704,A -85,B 0,C 180,E1 20447.34,E2 20447.34} C_VEL
LIN {X 0,Y 440.831,Z 1050.874,A -85,B 0,C 180,E1 20443.778,E2 20443.778} C_VEL
LIN {X 0,Y 440.282,Z 1056.093,A -85,B 0,C 180,E1 20440.865,E2 20440.865} C_VEL
LIN {X 0,Y 440.037,Z 1059.76,A -85,B 0,C 180,E1 20438.23,E2 20438.23} C_VEL
LIN {X 0,Y 439.923,Z 1062.574,A -85,B 0,C 180,E1 20435.422,E2 20435.422} C_VEL
LIN {X 0,Y 439.907,Z 1064.425,A -85,B 0,C 180,E1 20432.084,E2 20432.084} C_VEL
LIN {X 0,Y 439.908,Z 1064.646,A -85,B 0,C 180,E1 20429.219,E2 20429.219} C_VEL
LIN {X 0,Y 439.911,Z 1063.831,A -85,B 0,C 180,E1 20426.612,E2 20426.612} C_VEL
LIN {X 0,Y 439.937,Z 1062.019,A -85,B 0,C 180,E1 20423.999,E2 20423.999} C_VEL
LIN {X 0,Y 440.055,Z 1059.2,A -85,B 0,C 180,E1 20421.375,E2 20421.375} C_VEL
LIN {X 0,Y 440.415,Z 1054.516,A -85,B 0,C 180,E1 20418.21,E2 20418.21} C_VEL
LIN {X 0,Y 441.153,Z 1048.118,A -85,B 0,C 180,E1 20415.026,E2 20415.026} C_VEL
LIN {X 0,Y 442.215,Z 1041.232,A -85,B 0,C 180,E1 20412.227,E2 20412.227} C_VEL
LIN {X 0,Y 443.77,Z 1033.072,A -85,B 0,C 180,E1 20409.421,E2 20409.421} C_VEL
LIN {X 0,Y 446.401,Z 1021.349,A -85,B 0,C 180,E1 20406.047,E2 20406.047} C_VEL
LIN {X 0,Y 449.094,Z 1010.604,A -85,B 0,C 180,E1 20403.416,E2 20403.416} C_VEL
LIN {X 0,Y 452.481,Z 998.257,A -85,B 0,C 180,E1 20400.767,E2 20400.767} C_VEL
LIN {X 0,Y 457.189,Z 981.859,A -85,B 0,C 180,E1 20397.749,E2 20397.749} C_VEL
LIN {X 0,Y 461.271,Z 968.07,A -85,B 0,C 180,E1 20395.545,E2 20395.545} C_VEL
LIN {X 0,Y 466.035,Z 952.236,A -85,B 0,C 180,E1 20393.307,E2 20393.307} C_VEL
LIN {X 0,Y 471.968,Z 932.086,A -85,B 0,C 180,E1 20390.852,E2 20390.852} C_VEL
LIN {X 0,Y 476.851,Z 915.123,A -85,B 0,C 180,E1 20389.06,E2 20389.06} C_VEL
LIN {X 0,Y 482.532,Z 894.819,A -85,B 0,C 180,E1 20387.182,E2 20387.182} C_VEL
LIN {X 0,Y 488.219,Z 872.812,A -85,B 0,C 180,E1 20385.457,E2 20385.457} C_VEL
LIN {X 0,Y 492.789,Z 853.87,A -85,B 0,C 180,E1 20384.171,E2 20384.171} C_VEL
LIN {X 0,Y 497.838,Z 831.322,A -85,B 0,C 180,E1 20382.854,E2 20382.854} C_VEL
LIN {X 0,Y 502.378,Z 807.902,A -85,B 0,C 180,E1 20381.724,E2 20381.724} C_VEL
LIN {X 0,Y 506.04,Z 786.474,A -85,B 0,C 180,E1 20380.863,E2 20380.863} C_VEL
LIN {X 0,Y 509.731,Z 761.345,A -85,B 0,C 180,E1 20380.042,E2 20380.042} C_VEL
LIN {X 0,Y 512.583,Z 735.621,A -85,B 0,C 180,E1 20379.419,E2 20379.419} C_VEL
LIN {X 0,Y 514.344,Z 713.125,A -85,B 0,C 180,E1 20379.003,E2 20379.003} C_VEL
LIN {X 0,Y 525.425,Z 479.628,A -85,B 0,C 180,E1 20375.443,E2 20375.443} C_VEL
LIN {X 0,Y 528.944,Z 405.214,A -85,B 0,C 180,E1 20374.286,E2 20374.286} C_VEL
LIN {X 0,Y 517.085,Z 385.59,A -85,B 0,C 180,E1 20371.929,E2 20371.929} C_VEL
LIN {X 0,Y 505.105,Z 367.289,A -85,B 0,C 180,E1 20369.305,E2 20369.305} C_VEL
LIN {X 0,Y 495.188,Z 353.177,A -85,B 0,C 180,E1 20366.892,E2 20366.892} C_VEL
LIN {X 0,Y 489.543,Z 345.558,A -85,B 0,C 180,E1 20365.399,E2 20365.399} C_VEL
LIN {X 0,Y 485.261,Z 340.3,A -85,B 0,C 180,E1 20364.208,E2 20364.208} C_VEL
LIN {X 0,Y 480.803,Z 334.835,A -85,B 0,C 180,E1 20362.886,E2 20362.886} C_VEL
LIN {X 0,Y 477.01,Z 330.098,A -85,B 0,C 180,E1 20361.682,E2 20361.682} C_VEL
LIN {X 0,Y 472.765,Z 325.468,A -85,B 0,C 180,E1 20360.263,E2 20360.263} C_VEL
LIN {X 0,Y 471.263,Z 323.416,A -85,B 0,C 180,E1 20359.716,E2 20359.716} C_VEL
LIN {X 0,Y 467.804,Z 319.914,A -85,B 0,C 180,E1 20358.442,E2 20358.442} C_VEL
LIN {X 0,Y 466.088,Z 317.377,A -85,B 0,C 180,E1 20357.736,E2 20357.736} C_VEL
LIN {X 0,Y 462.768,Z 314.463,A -85,B 0,C 180,E1 20356.378,E2 20356.378} C_VEL
LIN {X 0,Y 460.907,Z 311.193,A -85,B 0,C 180,E1 20355.476,E2 20355.476} C_VEL
LIN {X 0,Y 457.314,Z 308.653,A -85,B 0,C 180,E1 20353.788,E2 20353.788} C_VEL
LIN {X 0,Y 455.295,Z 305.326,A -85,B 0,C 180,E1 20352.622,E2 20352.622} C_VEL
LIN {X 0,Y 454.561,Z 304.424,A -85,B 0,C 180,E1 20352.191,E2 20352.191} C_VEL
LIN {X 0,Y 451.105,Z 302.148,A -85,B 0,C 180,E1 20350.085,E2 20350.085} C_VEL
LIN {X 0,Y 449.291,Z 299.156,A -85,B 0,C 180,E1 20348.64,E2 20348.64} C_VEL
LIN {X 0,Y 448.346,Z 297.845,A -85,B 0,C 180,E1 20347.819,E2 20347.819} C_VEL
LIN {X 0,Y 443.018,Z 293.306,A -85,B 0,C 180,E1 20339.741,E2 20339.741} C_VEL
LIN {X 0,Y 442.973,Z 293.254,A -85,B 0,C 180,E1 20337.413,E2 20337.413} C_VEL
LIN {X 0,Y 443.99,Z 294.828,A -85,B 0,C 180,E1 20334.054,E2 20334.054} C_VEL
LIN {X 0,Y 448.895,Z 298.335,A -85,B 0,C 180,E1 20328.542,E2 20328.542} C_VEL
LIN {X 0,Y 450.837,Z 301.85,A -85,B 0,C 180,E1 20326.925,E2 20326.925} C_VEL
LIN {X 0,Y 454.224,Z 304.298,A -85,B 0,C 180,E1 20324.814,E2 20324.814} C_VEL
LIN {X 0,Y 455.159,Z 304.96,A -85,B 0,C 180,E1 20324.291,E2 20324.291} C_VEL
LIN {X 0,Y 457.089,Z 308.391,A -85,B 0,C 180,E1 20323.151,E2 20323.151} C_VEL
LIN {X 0,Y 460.781,Z 311.148,A -85,B 0,C 180,E1 20321.398,E2 20321.398} C_VEL
LIN {X 0,Y 463.61,Z 315.438,A -85,B 0,C 180,E1 20320.076,E2 20320.076} C_VEL
LIN {X 0,Y 466.631,Z 317.972,A -85,B 0,C 180,E1 20318.867,E2 20318.867} C_VEL
LIN {X 0,Y 469.513,Z 321.979,A -85,B 0,C 180,E1 20317.724,E2 20317.724} C_VEL
LIN {X 0,Y 472.101,Z 324.332,A -85,B 0,C 180,E1 20316.807,E2 20316.807} C_VEL
LIN {X 0,Y 475.407,Z 328.523,A -85,B 0,C 180,E1 20315.655,E2 20315.655} C_VEL
LIN {X 0,Y 477.242,Z 330.412,A -85,B 0,C 180,E1 20315.061,E2 20315.061} C_VEL
LIN {X 0,Y 481.074,Z 335.032,A -85,B 0,C 180,E1 20313.856,E2 20313.856} C_VEL
LIN {X 0,Y 487.481,Z 343.055,A -85,B 0,C 180,E1 20311.984,E2 20311.984} C_VEL
LIN {X 0,Y 492.383,Z 349.118,A -85,B 0,C 180,E1 20310.665,E2 20310.665} C_VEL
LIN {X 0,Y 499.519,Z 358.324,A -85,B 0,C 180,E1 20308.873,E2 20308.873} C_VEL
LIN {X 0,Y 510.349,Z 372.932,A -85,B 0,C 180,E1 20306.394,E2 20306.394} C_VEL
LIN {X 0,Y 520.461,Z 388.47,A -85,B 0,C 180,E1 20304.265,E2 20304.265} C_VEL
LIN {X 0,Y 529.094,Z 402.631,A -85,B 0,C 180,E1 20302.575,E2 20302.575} C_VEL
LIN {X 0,Y 519.311,Z 605.301,A -85,B 0,C 180,E1 20299.479,E2 20299.479} C_VEL
LIN {X 0,Y 514.1,Z 713.342,A -85,B 0,C 180,E1 20297.818,E2 20297.818} C_VEL
LIN {X 0,Y 511.534,Z 741.469,A -85,B 0,C 180,E1 20297.231,E2 20297.231} C_VEL
LIN {X 0,Y 508.831,Z 763.189,A -85,B 0,C 180,E1 20296.621,E2 20296.621} C_VEL
LIN {X 0,Y 505.845,Z 783.17,A -85,B 0,C 180,E1 20295.932,E2 20295.932} C_VEL
LIN {X 0,Y 501.79,Z 806.727,A -85,B 0,C 180,E1 20294.95,E2 20294.95} C_VEL
LIN {X 0,Y 497.083,Z 829.766,A -85,B 0,C 180,E1 20293.769,E2 20293.769} C_VEL
LIN {X 0,Y 492.666,Z 849.367,A -85,B 0,C 180,E1 20292.593,E2 20292.593} C_VEL
LIN {X 0,Y 487.284,Z 871.574,A -85,B 0,C 180,E1 20291.043,E2 20291.043} C_VEL
LIN {X 0,Y 481.599,Z 892.746,A -85,B 0,C 180,E1 20289.289,E2 20289.289} C_VEL
LIN {X 0,Y 476.663,Z 910.324,A -85,B 0,C 180,E1 20287.62,E2 20287.62} C_VEL
LIN {X 0,Y 470.943,Z 930.066,A -85,B 0,C 180,E1 20285.473,E2 20285.473} C_VEL
LIN {X 0,Y 465.527,Z 947.857,A -85,B 0,C 180,E1 20283.209,E2 20283.209} C_VEL
LIN {X 0,Y 461.009,Z 962.784,A -85,B 0,C 180,E1 20281.049,E2 20281.049} C_VEL
LIN {X 0,Y 456.035,Z 979.507,A -85,B 0,C 180,E1 20278.268,E2 20278.268} C_VEL
LIN {X 0,Y 452.129,Z 992.843,A -85,B 0,C 180,E1 20275.687,E2 20275.687} C_VEL
LIN {X 0,Y 448.867,Z 1004.686,A -85,B 0,C 180,E1 20273.074,E2 20273.074} C_VEL
LIN {X 0,Y 446.056,Z 1015.869,A -85,B 0,C 180,E1 20270.239,E2 20270.239} C_VEL
LIN {X 0,Y 444.302,Z 1019.142,A -85,B 0,C 180,E1 20269.358,E2 20269.358} C_VEL
LIN {X 0,Y 436.396,Z 1027.534,A -85,B 0,C 180,E1 20267.033,E2 20267.033} C_VEL
LIN {X 0,Y 435.173,Z 1029.952,A -85,B 0,C 180,E1 20266.234,E2 20266.234} C_VEL
LIN {X 0,Y 433.617,Z 1038.24,A -85,B 0,C 180,E1 20262.925,E2 20262.925} C_VEL
LIN {X 0,Y 432.788,Z 1043.885,A -85,B 0,C 180,E1 20260.194,E2 20260.194} C_VEL
LIN {X 0,Y 432.281,Z 1048.489,A -85,B 0,C 180,E1 20257.442,E2 20257.442} C_VEL
LIN {X 0,Y 432.008,Z 1052.679,A -85,B 0,C 180,E1 20254.114,E2 20254.114} C_VEL
LIN {X 0,Y 431.928,Z 1055.087,A -85,B 0,C 180,E1 20250.928,E2 20250.928} C_VEL
LIN {X 0,Y 431.904,Z 1056.073,A -85,B 0,C 180,E1 20248.275,E2 20248.275} C_VEL
LIN {X 0,Y 431.906,Z 1056.087,A -85,B 0,C 180,E1 20245.618,E2 20245.618} C_VEL
LIN {X 0,Y 431.934,Z 1055.124,A -85,B 0,C 180,E1 20242.953,E2 20242.953} C_VEL
LIN {X 0,Y 432.024,Z 1052.624,A -85,B 0,C 180,E1 20239.622,E2 20239.622} C_VEL
LIN {X 0,Y 432.32,Z 1048.37,A -85,B 0,C 180,E1 20236.264,E2 20236.264} C_VEL
LIN {X 0,Y 432.864,Z 1043.677,A -85,B 0,C 180,E1 20233.462,E2 20233.462} C_VEL
LIN {X 0,Y 433.786,Z 1037.781,A -85,B 0,C 180,E1 20230.614,E2 20230.614} C_VEL
LIN {X 0,Y 435.642,Z 1028.472,A -85,B 0,C 180,E1 20226.982,E2 20226.982} C_VEL
LIN {X 0,Y 437.75,Z 1019.639,A -85,B 0,C 180,E1 20224.134,E2 20224.134} C_VEL
LIN {X 0,Y 440.431,Z 1009.763,A -85,B 0,C 180,E1 20221.379,E2 20221.379} C_VEL
LIN {X 0,Y 444.717,Z 995.32,A -85,B 0,C 180,E1 20217.953,E2 20217.953} C_VEL
LIN {X 0,Y 448.75,Z 982.615,A -85,B 0,C 180,E1 20215.377,E2 20215.377} C_VEL
LIN {X 0,Y 453.718,Z 967.537,A -85,B 0,C 180,E1 20212.697,E2 20212.697} C_VEL
LIN {X 0,Y 459.461,Z 950.119,A -85,B 0,C 180,E1 20210.06,E2 20210.06} C_VEL
LIN {X 0,Y 464.391,Z 935.205,A -85,B 0,C 180,E1 20208.084,E2 20208.084} C_VEL
LIN {X 0,Y 470.452,Z 916.638,A -85,B 0,C 180,E1 20205.921,E2 20205.921} C_VEL
LIN {X 0,Y 476.703,Z 896.303,A -85,B 0,C 180,E1 20203.905,E2 20203.905} C_VEL
LIN {X 0,Y 481.898,Z 878.651,A -85,B 0,C 180,E1 20202.383,E2 20202.383} C_VEL
LIN {X 0,Y 487.492,Z 858.499,A -85,B 0,C 180,E1 20200.867,E2 20200.867} C_VEL
LIN {X 0,Y 493.417,Z 834.827,A -85,B 0,C 180,E1 20199.367,E2 20199.367} C_VEL
LIN {X 0,Y 497.768,Z 815.605,A -85,B 0,C 180,E1 20198.334,E2 20198.334} C_VEL
LIN {X 0,Y 501.801,Z 795.669,A -85,B 0,C 180,E1 20197.414,E2 20197.414} C_VEL
LIN {X 0,Y 506.37,Z 769.501,A -85,B 0,C 180,E1 20196.429,E2 20196.429} C_VEL
LIN {X 0,Y 509.524,Z 746.853,A -85,B 0,C 180,E1 20195.759,E2 20195.759} C_VEL
LIN {X 0,Y 512.05,Z 724.325,A -85,B 0,C 180,E1 20195.242,E2 20195.242} C_VEL
LIN {X 0,Y 514.392,Z 690.144,A -85,B 0,C 180,E1 20194.663,E2 20194.663} C_VEL
LIN {X 0,Y 526.453,Z 462.214,A -85,B 0,C 180,E1 20191.158,E2 20191.158} C_VEL
LIN {X 0,Y 529.323,Z 408.799,A -85,B 0,C 180,E1 20190.321,E2 20190.321} C_VEL
LIN {X 0,Y 519.36,Z 392.87,A -85,B 0,C 180,E1 20188.081,E2 20188.081} C_VEL
LIN {X 0,Y 511.186,Z 380.851,A -85,B 0,C 180,E1 20186.08,E2 20186.08} C_VEL
LIN {X 0,Y 502.515,Z 369.404,A -85,B 0,C 180,E1 20183.762,E2 20183.762} C_VEL
LIN {X 0,Y 496.397,Z 361.322,A -85,B 0,C 180,E1 20181.941,E2 20181.941} C_VEL
LIN {X 0,Y 491.479,Z 355.352,A -85,B 0,C 180,E1 20180.359,E2 20180.359} C_VEL
LIN {X 0,Y 487.218,Z 350.018,A -85,B 0,C 180,E1 20178.858,E2 20178.858} C_VEL
LIN {X 0,Y 483.397,Z 345.214,A -85,B 0,C 180,E1 20177.391,E2 20177.391} C_VEL
LIN {X 0,Y 479.018,Z 340.375,A -85,B 0,C 180,E1 20175.559,E2 20175.559} C_VEL
LIN {X 0,Y 477.653,Z 338.499,A -85,B 0,C 180,E1 20174.921,E2 20174.921} C_VEL
LIN {X 0,Y 474.282,Z 335.126,A -85,B 0,C 180,E1 20173.285,E2 20173.285} C_VEL
LIN {X 0,Y 472.617,Z 332.476,A -85,B 0,C 180,E1 20172.338,E2 20172.338} C_VEL
LIN {X 0,Y 469.009,Z 329.341,A -85,B 0,C 180,E1 20170.192,E2 20170.192} C_VEL
LIN {X 0,Y 467.284,Z 326.221,A -85,B 0,C 180,E1 20168.863,E2 20168.863} C_VEL
LIN {X 0,Y 463.431,Z 323.265,A -85,B 0,C 180,E1 20165.448,E2 20165.448} C_VEL
LIN {X 0,Y 461.757,Z 320.094,A -85,B 0,C 180,E1 20162.855,E2 20162.855} C_VEL
LIN {X 0,Y 460.576,Z 319.256,A -85,B 0,C 180,E1 20159.129,E2 20159.129} C_VEL
LIN {X 0,Y 461.674,Z 319.972,A -85,B 0,C 180,E1 20154.407,E2 20154.407} C_VEL
LIN {X 0,Y 462.202,Z 320.971,A -85,B 0,C 180,E1 20153.416,E2 20153.416} C_VEL
LIN {X 0,Y 464.799,Z 324.785,A -85,B 0,C 180,E1 20150.215,E2 20150.215} C_VEL
LIN {X 0,Y 467.55,Z 326.546,A -85,B 0,C 180,E1 20148.027,E2 20148.027} C_VEL
LIN {X 0,Y 469.686,Z 330.107,A -85,B 0,C 180,E1 20146.457,E2 20146.457} C_VEL
LIN {X 0,Y 473.031,Z 333.001,A -85,B 0,C 180,E1 20144.522,E2 20144.522} C_VEL
LIN {X 0,Y 475.704,Z 336.894,A -85,B 0,C 180,E1 20143.075,E2 20143.075} C_VEL
LIN {X 0,Y 478.417,Z 339.315,A -85,B 0,C 180,E1 20141.824,E2 20141.824} C_VEL
LIN {X 0,Y 481.901,Z 343.792,A -85,B 0,C 180,E1 20140.295,E2 20140.295} C_VEL
LIN {X 0,Y 483.544,Z 345.518,A -85,B 0,C 180,E1 20139.64,E2 20139.64} C_VEL
LIN {X 0,Y 487.314,Z 350.183,A -85,B 0,C 180,E1 20138.199,E2 20138.199} C_VEL
LIN {X 0,Y 493.419,Z 357.802,A -85,B 0,C 180,E1 20136.091,E2 20136.091} C_VEL
LIN {X 0,Y 499.495,Z 366.076,A -85,B 0,C 180,E1 20134.19,E2 20134.19} C_VEL
LIN {X 0,Y 507.279,Z 377.01,A -85,B 0,C 180,E1 20131.991,E2 20131.991} C_VEL
LIN {X 0,Y 514.995,Z 388.587,A -85,B 0,C 180,E1 20130.003,E2 20130.003} C_VEL
LIN {X 0,Y 524.068,Z 402.734,A -85,B 0,C 180,E1 20127.87,E2 20127.87} C_VEL
LIN {X 0,Y 529.373,Z 411.829,A -85,B 0,C 180,E1 20126.693,E2 20126.693} C_VEL
LIN {X 0,Y 517.2,Z 637.889,A -85,B 0,C 180,E1 20123.215,E2 20123.215} C_VEL
LIN {X 0,Y 512.756,Z 720.179,A -85,B 0,C 180,E1 20121.93,E2 20121.93} C_VEL
LIN {X 0,Y 509.921,Z 748.305,A -85,B 0,C 180,E1 20121.344,E2 20121.344} C_VEL
LIN {X 0,Y 507.068,Z 769.072,A -85,B 0,C 180,E1 20120.773,E2 20120.773} C_VEL
LIN {X 0,Y 503.66,Z 789.87,A -85,B 0,C 180,E1 20120.067,E2 20120.067} C_VEL
LIN {X 0,Y 499.06,Z 814.189,A -85,B 0,C 180,E1 20119.054,E2 20119.054} C_VEL
LIN {X 0,Y 493.986,Z 836.922,A -85,B 0,C 180,E1 20117.888,E2 20117.888} C_VEL
LIN {X 0,Y 489.136,Z 856.721,A -85,B 0,C 180,E1 20116.696,E2 20116.696} C_VEL
LIN {X 0,Y 483.18,Z 879.199,A -85,B 0,C 180,E1 20115.116,E2 20115.116} C_VEL
LIN {X 0,Y 477.205,Z 899.635,A -85,B 0,C 180,E1 20113.413,E2 20113.413} C_VEL
LIN {X 0,Y 471.795,Z 917.366,A -85,B 0,C 180,E1 20111.718,E2 20111.718} C_VEL
LIN {X 0,Y 465.423,Z 937.612,A -85,B 0,C 180,E1 20109.487,E2 20109.487} C_VEL
LIN {X 0,Y 459.639,Z 955.247,A -85,B 0,C 180,E1 20107.211,E2 20107.211} C_VEL
LIN {X 0,Y 454.752,Z 970.166,A -85,B 0,C 180,E1 20105.021,E2 20105.021} C_VEL
LIN {X 0,Y 449.239,Z 987.224,A -85,B 0,C 180,E1 20102.137,E2 20102.137} C_VEL
LIN {X 0,Y 445.003,Z 1000.715,A -85,B 0,C 180,E1 20099.477,E2 20099.477} C_VEL
LIN {X 0,Y 441.461,Z 1012.666,A -85,B 0,C 180,E1 20096.79,E2 20096.79} C_VEL
LIN {X 0,Y 437.995,Z 1025.529,A -85,B 0,C 180,E1 20093.404,E2 20093.404} C_VEL
LIN {X 0,Y 435.805,Z 1034.713,A -85,B 0,C 180,E1 20090.551,E2 20090.551} C_VEL
LIN {X 0,Y 434.147,Z 1042.989,A -85,B 0,C 180,E1 20087.542,E2 20087.542} C_VEL
LIN {X 0,Y 432.905,Z 1050.828,A -85,B 0,C 180,E1 20084.035,E2 20084.035} C_VEL
LIN {X 0,Y 432.329,Z 1055.832,A -85,B 0,C 180,E1 20081.202,E2 20081.202} C_VEL
LIN {X 0,Y 432.045,Z 1059.701,A -85,B 0,C 180,E1 20078.384,E2 20078.384} C_VEL
LIN {X 0,Y 431.923,Z 1062.46,A -85,B 0,C 180,E1 20075.58,E2 20075.58} C_VEL
LIN {X 0,Y 431.908,Z 1064.326,A -85,B 0,C 180,E1 20072.256,E2 20072.256} C_VEL
LIN {X 0,Y 431.908,Z 1064.566,A -85,B 0,C 180,E1 20069.204,E2 20069.204} C_VEL
LIN {X 0,Y 431.911,Z 1063.745,A -85,B 0,C 180,E1 20066.549,E2 20066.549} C_VEL
LIN {X 0,Y 431.942,Z 1061.928,A -85,B 0,C 180,E1 20063.887,E2 20063.887} C_VEL
LIN {X 0,Y 432.063,Z 1059.062,A -85,B 0,C 180,E1 20061.181,E2 20061.181} C_VEL
LIN {X 0,Y 432.484,Z 1054.185,A -85,B 0,C 180,E1 20057.855,E2 20057.855} C_VEL
LIN {X 0,Y 433.288,Z 1047.692,A -85,B 0,C 180,E1 20054.61,E2 20054.61} C_VEL
LIN {X 0,Y 434.373,Z 1041.104,A -85,B 0,C 180,E1 20051.895,E2 20051.895} C_VEL
LIN {X 0,Y 436.117,Z 1032.524,A -85,B 0,C 180,E1 20048.903,E2 20048.903} C_VEL
LIN {X 0,Y 438.896,Z 1020.801,A -85,B 0,C 180,E1 20045.504,E2 20045.504} C_VEL
LIN {X 0,Y 441.655,Z 1010.435,A -85,B 0,C 180,E1 20042.932,E2 20042.932} C_VEL
LIN {X 0,Y 445.198,Z 998.075,A -85,B 0,C 180,E1 20040.241,E2 20040.241} C_VEL
LIN {X 0,Y 449.906,Z 982.432,A -85,B 0,C 180,E1 20037.313,E2 20037.313} C_VEL
LIN {X 0,Y 454.432,Z 967.77,A -85,B 0,C 180,E1 20034.937,E2 20034.937} C_VEL
LIN {X 0,Y 459.656,Z 951.089,A -85,B 0,C 180,E1 20032.56,E2 20032.56} C_VEL
LIN {X 0,Y 465.538,Z 931.816,A -85,B 0,C 180,E1 20030.205,E2 20030.205} C_VEL
LIN {X 0,Y 470.553,Z 915.012,A -85,B 0,C 180,E1 20028.416,E2 20028.416} C_VEL
LIN {X 0,Y 476.496,Z 894.508,A -85,B 0,C 180,E1 20026.506,E2 20026.506} C_VEL
LIN {X 0,Y 482.322,Z 872.671,A -85,B 0,C 180,E1 20024.786,E2 20024.786} C_VEL
LIN {X 0,Y 487.099,Z 853.474,A -85,B 0,C 180,E1 20023.478,E2 20023.478} C_VEL
LIN {X 0,Y 492.541,Z 829.815,A -85,B 0,C 180,E1 20022.099,E2 20022.099} C_VEL
LIN {X 0,Y 497.116,Z 806.658,A -85,B 0,C 180,E1 20020.991,E2 20020.991} C_VEL
LIN {X 0,Y 500.709,Z 786.107,A -85,B 0,C 180,E1 20020.167,E2 20020.167} C_VEL
LIN {X 0,Y 504.538,Z 760.57,A -85,B 0,C 180,E1 20019.336,E2 20019.336} C_VEL
LIN {X 0,Y 507.41,Z 735.271,A -85,B 0,C 180,E1 20018.725,E2 20018.725} C_VEL
LIN {X 0,Y 509.216,Z 712.688,A -85,B 0,C 180,E1 20018.308,E2 20018.308} C_VEL
LIN {X 0,Y 520.668,Z 479.327,A -85,B 0,C 180,E1 20014.731,E2 20014.731} C_VEL
LIN {X 0,Y 524.153,Z 409.159,A -85,B 0,C 180,E1 20013.642,E2 20013.642} C_VEL
LIN {X 0,Y 513.24,Z 391.067,A -85,B 0,C 180,E1 20011.409,E2 20011.409} C_VEL
LIN {X 0,Y 501.901,Z 373.521,A -85,B 0,C 180,E1 20008.856,E2 20008.856} C_VEL
LIN {X 0,Y 492.242,Z 359.632,A -85,B 0,C 180,E1 20006.447,E2 20006.447} C_VEL
LIN {X 0,Y 487.079,Z 352.58,A -85,B 0,C 180,E1 20005.049,E2 20005.049} C_VEL
LIN {X 0,Y 482.856,Z 347.352,A -85,B 0,C 180,E1 20003.849,E2 20003.849} C_VEL
LIN {X 0,Y 478.555,Z 342.017,A -85,B 0,C 180,E1 20002.545,E2 20002.545} C_VEL
LIN {X 0,Y 474.038,Z 336.541,A -85,B 0,C 180,E1 20001.078,E2 20001.078} C_VEL
LIN {X 0,Y 470.348,Z 332.113,A -85,B 0,C 180,E1 19999.788,E2 19999.788} C_VEL
LIN {X 0,Y 469.159,Z 330.736,A -85,B 0,C 180,E1 19999.354,E2 19999.354} C_VEL
LIN {X 0,Y 465.716,Z 326.946,A -85,B 0,C 180,E1 19998.041,E2 19998.041} C_VEL
LIN {X 0,Y 464.53,Z 325.082,A -85,B 0,C 180,E1 19997.539,E2 19997.539} C_VEL
LIN {X 0,Y 461.117,Z 321.998,A -85,B 0,C 180,E1 19996.115,E2 19996.115} C_VEL
LIN {X 0,Y 459.136,Z 318.81,A -85,B 0,C 180,E1 19995.149,E2 19995.149} C_VEL
LIN {X 0,Y 455.532,Z 315.933,A -85,B 0,C 180,E1 19993.39,E2 19993.39} C_VEL
LIN {X 0,Y 453.378,Z 312.305,A -85,B 0,C 180,E1 19992.094,E2 19992.094} C_VEL
LIN {X 0,Y 449.95,Z 310.035,A -85,B 0,C 180,E1 19989.982,E2 19989.982} C_VEL
LIN {X 0,Y 448.071,Z 307.029,A -85,B 0,C 180,E1 19988.469,E2 19988.469} C_VEL
LIN {X 0,Y 447.373,Z 305.841,A -85,B 0,C 180,E1 19987.836,E2 19987.836} C_VEL
LIN {X 0,Y 442.023,Z 301.222,A -85,B 0,C 180,E1 19979.611,E2 19979.611} C_VEL
LIN {X 0,Y 442.012,Z 301.228,A -85,B 0,C 180,E1 19977.277,E2 19977.277} C_VEL
LIN {X 0,Y 443.217,Z 303.099,A -85,B 0,C 180,E1 19973.653,E2 19973.653} C_VEL
LIN {X 0,Y 447.746,Z 306.208,A -85,B 0,C 180,E1 19968.666,E2 19968.666} C_VEL
LIN {X 0,Y 449.522,Z 309.554,A -85,B 0,C 180,E1 19967.148,E2 19967.148} C_VEL
LIN {X 0,Y 453.055,Z 312.184,A -85,B 0,C 180,E1 19964.905,E2 19964.905} C_VEL
LIN {X 0,Y 453.747,Z 312.812,A -85,B 0,C 180,E1 19964.503,E2 19964.503} C_VEL
LIN {X 0,Y 455.892,Z 316.352,A -85,B 0,C 180,E1 19963.237,E2 19963.237} C_VEL
LIN {X 0,Y 459.534,Z 319.363,A -85,B 0,C 180,E1 19961.477,E2 19961.477} C_VEL
LIN {X 0,Y 462.205,Z 323.25,A -85,B 0,C 180,E1 19960.225,E2 19960.225} C_VEL
LIN {X 0,Y 464.924,Z 325.64,A -85,B 0,C 180,E1 19959.116,E2 19959.116} C_VEL
LIN {X 0,Y 467.936,Z 329.684,A -85,B 0,C 180,E1 19957.909,E2 19957.909} C_VEL
LIN {X 0,Y 470.264,Z 331.899,A -85,B 0,C 180,E1 19957.068,E2 19957.068} C_VEL
LIN {X 0,Y 473.777,Z 336.233,A -85,B 0,C 180,E1 19955.831,E2 19955.831} C_VEL
LIN {X 0,Y 475.404,Z 338.089,A -85,B 0,C 180,E1 19955.29,E2 19955.29} C_VEL
LIN {X 0,Y 480.28,Z 344.114,A -85,B 0,C 180,E1 19953.743,E2 19953.743} C_VEL
LIN {X 0,Y 485.352,Z 350.475,A -85,B 0,C 180,E1 19952.251,E2 19952.251} C_VEL
LIN {X 0,Y 490.303,Z 356.67,A -85,B 0,C 180,E1 19950.897,E2 19950.897} C_VEL
LIN {X 0,Y 497.689,Z 366.411,A -85,B 0,C 180,E1 19949.014,E2 19949.014} C_VEL
LIN {X 0,Y 507.653,Z 380.018,A -85,B 0,C 180,E1 19946.699,E2 19946.699} C_VEL
LIN {X 0,Y 518.5,Z 396.934,A -85,B 0,C 180,E1 19944.381,E2 19944.381} C_VEL
LIN {X 0,Y 524.247,Z 406.793,A -85,B 0,C 180,E1 19943.224,E2 19943.224} C_VEL
LIN {X 0,Y 514.014,Z 611.922,A -85,B 0,C 180,E1 19940.076,E2 19940.076} C_VEL
LIN {X 0,Y 508.935,Z 713.519,A -85,B 0,C 180,E1 19938.503,E2 19938.503} C_VEL
LIN {X 0,Y 506.292,Z 741.672,A -85,B 0,C 180,E1 19937.914,E2 19937.914} C_VEL
LIN {X 0,Y 503.544,Z 763.161,A -85,B 0,C 180,E1 19937.309,E2 19937.309} C_VEL
LIN {X 0,Y 500.571,Z 782.523,A -85,B 0,C 180,E1 19936.642,E2 19936.642} C_VEL
LIN {X 0,Y 496.368,Z 806.315,A -85,B 0,C 180,E1 19935.652,E2 19935.652} C_VEL
LIN {X 0,Y 491.371,Z 830.148,A -85,B 0,C 180,E1 19934.427,E2 19934.427} C_VEL
LIN {X 0,Y 487.002,Z 848.957,A -85,B 0,C 180,E1 19933.294,E2 19933.294} C_VEL
LIN {X 0,Y 481.618,Z 870.474,A -85,B 0,C 180,E1 19931.792,E2 19931.792} C_VEL
LIN {X 0,Y 475.731,Z 891.856,A -85,B 0,C 180,E1 19930.027,E2 19930.027} C_VEL
LIN {X 0,Y 470.601,Z 909.523,A -85,B 0,C 180,E1 19928.346,E2 19928.346} C_VEL
LIN {X 0,Y 464.863,Z 928.677,A -85,B 0,C 180,E1 19926.264,E2 19926.264} C_VEL
LIN {X 0,Y 459.017,Z 947.272,A -85,B 0,C 180,E1 19923.893,E2 19923.893} C_VEL
LIN {X 0,Y 454.336,Z 962.096,A -85,B 0,C 180,E1 19921.734,E2 19921.734} C_VEL
LIN {X 0,Y 449.278,Z 978.399,A -85,B 0,C 180,E1 19919.023,E2 19919.023} C_VEL
LIN {X 0,Y 444.955,Z 992.474,A -85,B 0,C 180,E1 19916.276,E2 19916.276} C_VEL
LIN {X 0,Y 441.663,Z 1003.764,A -85,B 0,C 180,E1 19913.764,E2 19913.764} C_VEL
LIN {X 0,Y 438.486,Z 1015.776,A -85,B 0,C 180,E1 19910.698,E2 19910.698} C_VEL
LIN {X 0,Y 435.942,Z 1026.234,A -85,B 0,C 180,E1 19907.485,E2 19907.485} C_VEL
LIN {X 0,Y 435.173,Z 1029.952,A -85,B 0,C 180,E1 19906.234,E2 19906.234} C_VEL
LIN {X 0,Y 433.67,Z 1032.661,A -85,B 0,C 180,E1 19905.295,E2 19905.295} C_VEL
LIN {X 0,Y 426.174,Z 1039.363,A -85,B 0,C 180,E1 19902.711,E2 19902.711} C_VEL
LIN {X 0,Y 425.286,Z 1041.117,A -85,B 0,C 180,E1 19901.931,E2 19901.931} C_VEL
LIN {X 0,Y 424.455,Z 1047.2,A -85,B 0,C 180,E1 19898.535,E2 19898.535} C_VEL
LIN {X 0,Y 424.101,Z 1051.101,A -85,B 0,C 180,E1 19895.683,E2 19895.683} C_VEL
LIN {X 0,Y 423.956,Z 1053.802,A -85,B 0,C 180,E1 19892.974,E2 19892.974} C_VEL
LIN {X 0,Y 423.935,Z 1055.657,A -85,B 0,C 180,E1 19890,E2 19890} C_VEL
LIN {X 0,Y 423.9,Z 1056.338,A -85,B 0,C 180,E1 19886.619,E2 19886.619} C_VEL
LIN {X 0,Y 423.921,Z 1055.52,A -85,B 0,C 180,E1 19883.499,E2 19883.499} C_VEL
LIN {X 0,Y 423.967,Z 1053.784,A -85,B 0,C 180,E1 19880.772,E2 19880.772} C_VEL
LIN {X 0,Y 424.122,Z 1051.048,A -85,B 0,C 180,E1 19878.026,E2 19878.026} C_VEL
LIN {X 0,Y 424.554,Z 1046.794,A -85,B 0,C 180,E1 19874.932,E2 19874.932} C_VEL
LIN {X 0,Y 425.518,Z 1040.201,A -85,B 0,C 180,E1 19871.363,E2 19871.363} C_VEL
LIN {X 0,Y 426.816,Z 1033.406,A -85,B 0,C 180,E1 19868.42,E2 19868.42} C_VEL
LIN {X 0,Y 428.705,Z 1025.329,A -85,B 0,C 180,E1 19865.471,E2 19865.471} C_VEL
LIN {X 0,Y 431.957,Z 1013.322,A -85,B 0,C 180,E1 19861.822,E2 19861.822} C_VEL
LIN {X 0,Y 435.26,Z 1002.455,A -85,B 0,C 180,E1 19859.031,E2 19859.031} C_VEL
LIN {X 0,Y 439.717,Z 988.828,A -85,B 0,C 180,E1 19855.987,E2 19855.987} C_VEL
LIN {X 0,Y 444.844,Z 973.623,A -85,B 0,C 180,E1 19853.12,E2 19853.12} C_VEL
LIN {X 0,Y 449.626,Z 959.78,A -85,B 0,C 180,E1 19850.834,E2 19850.834} C_VEL
LIN {X 0,Y 455.667,Z 942.452,A -85,B 0,C 180,E1 19848.327,E2 19848.327} C_VEL
LIN {X 0,Y 461.837,Z 924.099,A -85,B 0,C 180,E1 19846.068,E2 19846.068} C_VEL
LIN {X 0,Y 467.456,Z 907.003,A -85,B 0,C 180,E1 19844.229,E2 19844.229} C_VEL
LIN {X 0,Y 474.151,Z 885.777,A -85,B 0,C 180,E1 19842.253,E2 19842.253} C_VEL
LIN {X 0,Y 479.92,Z 865.875,A -85,B 0,C 180,E1 19840.679,E2 19840.679} C_VEL
LIN {X 0,Y 485.048,Z 846.867,A -85,B 0,C 180,E1 19839.373,E2 19839.373} C_VEL
LIN {X 0,Y 490.95,Z 823.115,A -85,B 0,C 180,E1 19837.985,E2 19837.985} C_VEL
LIN {X 0,Y 495.754,Z 800.575,A -85,B 0,C 180,E1 19836.899,E2 19836.899} C_VEL
LIN {X 0,Y 499.681,Z 779.691,A -85,B 0,C 180,E1 19836.058,E2 19836.058} C_VEL
LIN {X 0,Y 503.755,Z 754.157,A -85,B 0,C 180,E1 19835.225,E2 19835.225} C_VEL
LIN {X 0,Y 506.77,Z 729.199,A -85,B 0,C 180,E1 19834.619,E2 19834.619} C_VEL
LIN {X 0,Y 508.705,Z 706.721,A -85,B 0,C 180,E1 19834.201,E2 19834.201} C_VEL
LIN {X 0,Y 521.545,Z 472.941,A -85,B 0,C 180,E1 19830.586,E2 19830.586} C_VEL
LIN {X 0,Y 524.836,Z 412.971,A -85,B 0,C 180,E1 19829.636,E2 19829.636} C_VEL
LIN {X 0,Y 514.963,Z 397.256,A -85,B 0,C 180,E1 19827.336,E2 19827.336} C_VEL
LIN {X 0,Y 508.277,Z 387.326,A -85,B 0,C 180,E1 19825.645,E2 19825.645} C_VEL
LIN {X 0,Y 498.241,Z 373.703,A -85,B 0,C 180,E1 19822.85,E2 19822.85} C_VEL
LIN {X 0,Y 490.18,Z 363.397,A -85,B 0,C 180,E1 19820.29,E2 19820.29} C_VEL
LIN {X 0,Y 485.164,Z 357.258,A -85,B 0,C 180,E1 19818.505,E2 19818.505} C_VEL
LIN {X 0,Y 480.851,Z 351.916,A -85,B 0,C 180,E1 19816.801,E2 19816.801} C_VEL
LIN {X 0,Y 477.152,Z 347.534,A -85,B 0,C 180,E1 19815.185,E2 19815.185} C_VEL
LIN {X 0,Y 476.175,Z 346.205,A -85,B 0,C 180,E1 19814.719,E2 19814.719} C_VEL
LIN {X 0,Y 472.854,Z 342.818,A -85,B 0,C 180,E1 19813.077,E2 19813.077} C_VEL
LIN {X 0,Y 471.211,Z 340.224,A -85,B 0,C 180,E1 19812.127,E2 19812.127} C_VEL
LIN {X 0,Y 467.594,Z 336.903,A -85,B 0,C 180,E1 19809.912,E2 19809.912} C_VEL
LIN {X 0,Y 465.98,Z 334.026,A -85,B 0,C 180,E1 19808.639,E2 19808.639} C_VEL
LIN {X 0,Y 462.248,Z 330.991,A -85,B 0,C 180,E1 19805.213,E2 19805.213} C_VEL
LIN {X 0,Y 460.714,Z 327.984,A -85,B 0,C 180,E1 19802.737,E2 19802.737} C_VEL
LIN {X 0,Y 459.584,Z 327.199,A -85,B 0,C 180,E1 19798.878,E2 19798.878} C_VEL
LIN {X 0,Y 460.701,Z 327.929,A -85,B 0,C 180,E1 19794.395,E2 19794.395} C_VEL
LIN {X 0,Y 461.56,Z 329.852,A -85,B 0,C 180,E1 19792.827,E2 19792.827} C_VEL
LIN {X 0,Y 464.384,Z 333.168,A -85,B 0,C 180,E1 19789.705,E2 19789.705} C_VEL
LIN {X 0,Y 466.327,Z 334.45,A -85,B 0,C 180,E1 19788.184,E2 19788.184} C_VEL
LIN {X 0,Y 468.532,Z 338.013,A -85,B 0,C 180,E1 19786.549,E2 19786.549} C_VEL
LIN {X 0,Y 471.635,Z 340.782,A -85,B 0,C 180,E1 19784.722,E2 19784.722} C_VEL
LIN {X 0,Y 474.504,Z 344.826,A -85,B 0,C 180,E1 19783.157,E2 19783.157} C_VEL
LIN {X 0,Y 476.873,Z 346.997,A -85,B 0,C 180,E1 19782.048,E2 19782.048} C_VEL
LIN {X 0,Y 480.525,Z 351.616,A -85,B 0,C 180,E1 19780.427,E2 19780.427} C_VEL
LIN {X 0,Y 481.994,Z 353.338,A -85,B 0,C 180,E1 19779.825,E2 19779.825} C_VEL
LIN {X 0,Y 485.897,Z 358.022,A -85,B 0,C 180,E1 19778.323,E2 19778.323} C_VEL
LIN {X 0,Y 491.773,Z 365.641,A -85,B 0,C 180,E1 19776.26,E2 19776.26} C_VEL
LIN {X 0,Y 497.345,Z 373.365,A -85,B 0,C 180,E1 19774.485,E2 19774.485} C_VEL
LIN {X 0,Y 505.416,Z 384.866,A -85,B 0,C 180,E1 19772.167,E2 19772.167} C_VEL
LIN {X 0,Y 515.035,Z 399.579,A -85,B 0,C 180,E1 19769.684,E2 19769.684} C_VEL
LIN {X 0,Y 524.129,Z 414.539,A -85,B 0,C 180,E1 19767.551,E2 19767.551} C_VEL
LIN {X 0,Y 524.906,Z 416.121,A -85,B 0,C 180,E1 19767.37,E2 19767.37} C_VEL
LIN {X 0,Y 512.418,Z 640.771,A -85,B 0,C 180,E1 19763.9,E2 19763.9} C_VEL
LIN {X 0,Y 507.976,Z 720.266,A -85,B 0,C 180,E1 19762.653,E2 19762.653} C_VEL
LIN {X 0,Y 505.067,Z 748.326,A -85,B 0,C 180,E1 19762.067,E2 19762.067} C_VEL
LIN {X 0,Y 502.134,Z 769.073,A -85,B 0,C 180,E1 19761.496,E2 19761.496} C_VEL
LIN {X 0,Y 498.553,Z 790.316,A -85,B 0,C 180,E1 19760.774,E2 19760.774} C_VEL
LIN {X 0,Y 493.565,Z 815.632,A -85,B 0,C 180,E1 19759.705,E2 19759.705} C_VEL
LIN {X 0,Y 488.601,Z 837.199,A -85,B 0,C 180,E1 19758.592,E2 19758.592} C_VEL
LIN {X 0,Y 483.611,Z 856.962,A -85,B 0,C 180,E1 19757.396,E2 19757.396} C_VEL
LIN {X 0,Y 477.281,Z 879.966,A -85,B 0,C 180,E1 19755.763,E2 19755.763} C_VEL
LIN {X 0,Y 471.116,Z 900.348,A -85,B 0,C 180,E1 19754.047,E2 19754.047} C_VEL
LIN {X 0,Y 465.308,Z 918.707,A -85,B 0,C 180,E1 19752.268,E2 19752.268} C_VEL
LIN {X 0,Y 458.374,Z 939.725,A -85,B 0,C 180,E1 19749.891,E2 19749.891} C_VEL
LIN {X 0,Y 452.912,Z 955.779,A -85,B 0,C 180,E1 19747.781,E2 19747.781} C_VEL
LIN {X 0,Y 447.698,Z 971.07,A -85,B 0,C 180,E1 19745.499,E2 19745.499} C_VEL
LIN {X 0,Y 441.972,Z 987.959,A -85,B 0,C 180,E1 19742.577,E2 19742.577} C_VEL
LIN {X 0,Y 437.768,Z 1000.737,A -85,B 0,C 180,E1 19740.014,E2 19740.014} C_VEL
LIN {X 0,Y 434.059,Z 1012.676,A -85,B 0,C 180,E1 19737.285,E2 19737.285} C_VEL
LIN {X 0,Y 430.398,Z 1025.519,A -85,B 0,C 180,E1 19733.843,E2 19733.843} C_VEL
LIN {X 0,Y 428.071,Z 1034.693,A -85,B 0,C 180,E1 19730.939,E2 19730.939} C_VEL
LIN {X 0,Y 426.315,Z 1042.914,A -85,B 0,C 180,E1 19727.894,E2 19727.894} C_VEL
LIN {X 0,Y 424.959,Z 1050.956,A -85,B 0,C 180,E1 19724.209,E2 19724.209} C_VEL
LIN {X 0,Y 424.342,Z 1055.988,A -85,B 0,C 180,E1 19721.278,E2 19721.278} C_VEL
LIN {X 0,Y 424.048,Z 1059.803,A -85,B 0,C 180,E1 19718.406,E2 19718.406} C_VEL
LIN {X 0,Y 423.921,Z 1062.854,A -85,B 0,C 180,E1 19715.142,E2 19715.142} C_VEL
LIN {X 0,Y 423.904,Z 1064.32,A -85,B 0,C 180,E1 19711.892,E2 19711.892} C_VEL
LIN {X 0,Y 423.911,Z 1064.462,A -85,B 0,C 180,E1 19709.054,E2 19709.054} C_VEL
LIN {X 0,Y 423.912,Z 1063.59,A -85,B 0,C 180,E1 19706.349,E2 19706.349} C_VEL
LIN {X 0,Y 423.955,Z 1061.721,A -85,B 0,C 180,E1 19703.636,E2 19703.636} C_VEL
LIN {X 0,Y 424.113,Z 1058.519,A -85,B 0,C 180,E1 19700.638,E2 19700.638} C_VEL
LIN {X 0,Y 424.63,Z 1053.045,A -85,B 0,C 180,E1 19697.074,E2 19697.074} C_VEL
LIN {X 0,Y 425.438,Z 1047.263,A -85,B 0,C 180,E1 19694.179,E2 19694.179} C_VEL
LIN {X 0,Y 426.614,Z 1040.615,A -85,B 0,C 180,E1 19691.413,E2 19691.413} C_VEL
LIN {X 0,Y 428.714,Z 1031.147,A -85,B 0,C 180,E1 19688.089,E2 19688.089} C_VEL
LIN {X 0,Y 431.47,Z 1020.12,A -85,B 0,C 180,E1 19684.908,E2 19684.908} C_VEL
LIN {X 0,Y 434.415,Z 1009.682,A -85,B 0,C 180,E1 19682.294,E2 19682.294} C_VEL
LIN {X 0,Y 438.665,Z 995.71,A -85,B 0,C 180,E1 19679.242,E2 19679.242} C_VEL
LIN {X 0,Y 443.383,Z 980.664,A -85,B 0,C 180,E1 19676.461,E2 19676.461} C_VEL
LIN {X 0,Y 448.085,Z 966.1,A -85,B 0,C 180,E1 19674.099,E2 19674.099} C_VEL
LIN {X 0,Y 454.16,Z 947.351,A -85,B 0,C 180,E1 19671.46,E2 19671.46} C_VEL
LIN {X 0,Y 459.688,Z 929.915,A -85,B 0,C 180,E1 19669.357,E2 19669.357} C_VEL
LIN {X 0,Y 465.067,Z 912.517,A -85,B 0,C 180,E1 19667.515,E2 19667.515} C_VEL
LIN {X 0,Y 471.758,Z 889.778,A -85,B 0,C 180,E1 19665.449,E2 19665.449} C_VEL
LIN {X 0,Y 476.83,Z 871.263,A -85,B 0,C 180,E1 19664.007,E2 19664.007} C_VEL
LIN {X 0,Y 481.718,Z 852.167,A -85,B 0,C 180,E1 19662.711,E2 19662.711} C_VEL
LIN {X 0,Y 487.327,Z 828.188,A -85,B 0,C 180,E1 19661.328,E2 19661.328} C_VEL
LIN {X 0,Y 491.75,Z 806.403,A -85,B 0,C 180,E1 19660.286,E2 19660.286} C_VEL
LIN {X 0,Y 495.493,Z 785.519,A -85,B 0,C 180,E1 19659.448,E2 19659.448} C_VEL
LIN {X 0,Y 499.429,Z 759.733,A -85,B 0,C 180,E1 19658.614,E2 19658.614} C_VEL
LIN {X 0,Y 502.299,Z 735.085,A -85,B 0,C 180,E1 19658.021,E2 19658.021} C_VEL
LIN {X 0,Y 504.156,Z 712.359,A -85,B 0,C 180,E1 19657.6,E2 19657.6} C_VEL
LIN {X 0,Y 515.981,Z 479.277,A -85,B 0,C 180,E1 19654.01,E2 19654.01} C_VEL
LIN {X 0,Y 519.384,Z 413.131,A -85,B 0,C 180,E1 19652.979,E2 19652.979} C_VEL
LIN {X 0,Y 508.985,Z 395.787,A -85,B 0,C 180,E1 19650.78,E2 19650.78} C_VEL
LIN {X 0,Y 498.304,Z 379.09,A -85,B 0,C 180,E1 19648.298,E2 19648.298} C_VEL
LIN {X 0,Y 486.783,Z 362.296,A -85,B 0,C 180,E1 19645.293,E2 19645.293} C_VEL
LIN {X 0,Y 480.565,Z 354.496,A -85,B 0,C 180,E1 19643.514,E2 19643.514} C_VEL
LIN {X 0,Y 476.146,Z 349.003,A -85,B 0,C 180,E1 19642.145,E2 19642.145} C_VEL
LIN {X 0,Y 472.047,Z 343.923,A -85,B 0,C 180,E1 19640.781,E2 19640.781} C_VEL
LIN {X 0,Y 468.263,Z 339.242,A -85,B 0,C 180,E1 19639.425,E2 19639.425} C_VEL
LIN {X 0,Y 463.791,Z 334.192,A -85,B 0,C 180,E1 19637.697,E2 19637.697} C_VEL
LIN {X 0,Y 462.678,Z 332.594,A -85,B 0,C 180,E1 19637.222,E2 19637.222} C_VEL
LIN {X 0,Y 459.347,Z 329.358,A -85,B 0,C 180,E1 19635.789,E2 19635.789} C_VEL
LIN {X 0,Y 457.648,Z 326.551,A -85,B 0,C 180,E1 19634.94,E2 19634.94} C_VEL
LIN {X 0,Y 453.992,Z 323.475,A -85,B 0,C 180,E1 19633.112,E2 19633.112} C_VEL
LIN {X 0,Y 451.974,Z 320.094,A -85,B 0,C 180,E1 19631.873,E2 19631.873} C_VEL
LIN {X 0,Y 448.45,Z 317.544,A -85,B 0,C 180,E1 19629.627,E2 19629.627} C_VEL
LIN {X 0,Y 446.6,Z 314.226,A -85,B 0,C 180,E1 19628.044,E2 19628.044} C_VEL
LIN {X 0,Y 445.381,Z 313.256,A -85,B 0,C 180,E1 19626.963,E2 19626.963} C_VEL
LIN {X 0,Y 441.047,Z 309.164,A -85,B 0,C 180,E1 19619.61,E2 19619.61} C_VEL
LIN {X 0,Y 441.023,Z 309.143,A -85,B 0,C 180,E1 19617.401,E2 19617.401} C_VEL
LIN {X 0,Y 442.104,Z 310.889,A -85,B 0,C 180,E1 19613.898,E2 19613.898} C_VEL
LIN {X 0,Y 446.551,Z 314.043,A -85,B 0,C 180,E1 19608.832,E2 19608.832} C_VEL
LIN {X 0,Y 448.297,Z 317.359,A -85,B 0,C 180,E1 19607.309,E2 19607.309} C_VEL
LIN {X 0,Y 451.888,Z 320.069,A -85,B 0,C 180,E1 19604.996,E2 19604.996} C_VEL
LIN {X 0,Y 452.533,Z 321.049,A -85,B 0,C 180,E1 19604.592,E2 19604.592} C_VEL
LIN {X 0,Y 454.93,Z 324.532,A -85,B 0,C 180,E1 19603.2,E2 19603.2} C_VEL
LIN {X 0,Y 457.925,Z 326.983,A -85,B 0,C 180,E1 19601.74,E2 19601.74} C_VEL
LIN {X 0,Y 460.726,Z 330.978,A -85,B 0,C 180,E1 19600.409,E2 19600.409} C_VEL
LIN {X 0,Y 463.228,Z 333.28,A -85,B 0,C 180,E1 19599.367,E2 19599.367} C_VEL
LIN {X 0,Y 466.52,Z 337.535,A -85,B 0,C 180,E1 19598.037,E2 19598.037} C_VEL
LIN {X 0,Y 468.496,Z 339.543,A -85,B 0,C 180,E1 19597.309,E2 19597.309} C_VEL
LIN {X 0,Y 472.324,Z 344.093,A -85,B 0,C 180,E1 19595.951,E2 19595.951} C_VEL
LIN {X 0,Y 478.222,Z 351.526,A -85,B 0,C 180,E1 19594.021,E2 19594.021} C_VEL
LIN {X 0,Y 483.425,Z 358.138,A -85,B 0,C 180,E1 19592.466,E2 19592.466} C_VEL
LIN {X 0,Y 489.957,Z 366.357,A -85,B 0,C 180,E1 19590.673,E2 19590.673} C_VEL
LIN {X 0,Y 500.848,Z 381.263,A -85,B 0,C 180,E1 19587.958,E2 19587.958} C_VEL
LIN {X 0,Y 508.138,Z 391.972,A -85,B 0,C 180,E1 19586.296,E2 19586.296} C_VEL
LIN {X 0,Y 519.483,Z 410.461,A -85,B 0,C 180,E1 19583.894,E2 19583.894} C_VEL
LIN {X 0,Y 509.116,Z 611.661,A -85,B 0,C 180,E1 19580.791,E2 19580.791} C_VEL
LIN {X 0,Y 503.852,Z 713.59,A -85,B 0,C 180,E1 19579.205,E2 19579.205} C_VEL
LIN {X 0,Y 501.141,Z 741.747,A -85,B 0,C 180,E1 19578.613,E2 19578.613} C_VEL
LIN {X 0,Y 498.33,Z 763.131,A -85,B 0,C 180,E1 19578.011,E2 19578.011} C_VEL
LIN {X 0,Y 495.138,Z 783.332,A -85,B 0,C 180,E1 19577.312,E2 19577.312} C_VEL
LIN {X 0,Y 490.583,Z 808.157,A -85,B 0,C 180,E1 19576.263,E2 19576.263} C_VEL
LIN {X 0,Y 485.678,Z 830.73,A -85,B 0,C 180,E1 19575.089,E2 19575.089} C_VEL
LIN {X 0,Y 481.029,Z 850.125,A -85,B 0,C 180,E1 19573.909,E2 19573.909} C_VEL
LIN {X 0,Y 475.227,Z 872.509,A -85,B 0,C 180,E1 19572.321,E2 19572.321} C_VEL
LIN {X 0,Y 469.364,Z 892.936,A -85,B 0,C 180,E1 19570.602,E2 19570.602} C_VEL
LIN {X 0,Y 464.078,Z 910.517,A -85,B 0,C 180,E1 19568.907,E2 19568.907} C_VEL
LIN {X 0,Y 457.822,Z 930.59,A -85,B 0,C 180,E1 19566.678,E2 19566.678} C_VEL
LIN {X 0,Y 452.168,Z 947.89,A -85,B 0,C 180,E1 19564.429,E2 19564.429} C_VEL
LIN {X 0,Y 447.405,Z 962.401,A -85,B 0,C 180,E1 19562.285,E2 19562.285} C_VEL
LIN {X 0,Y 442.131,Z 978.669,A -85,B 0,C 180,E1 19559.539,E2 19559.539} C_VEL
LIN {X 0,Y 437.623,Z 992.728,A -85,B 0,C 180,E1 19556.75,E2 19556.75} C_VEL
LIN {X 0,Y 434.187,Z 1004.003,A -85,B 0,C 180,E1 19554.199,E2 19554.199} C_VEL
LIN {X 0,Y 430.72,Z 1016.439,A -85,B 0,C 180,E1 19550.947,E2 19550.947} C_VEL
LIN {X 0,Y 428.174,Z 1026.428,A -85,B 0,C 180,E1 19547.813,E2 19547.813} C_VEL
LIN {X 0,Y 426.492,Z 1034.225,A -85,B 0,C 180,E1 19544.945,E2 19544.945} C_VEL
LIN {X 0,Y 425.286,Z 1041.117,A -85,B 0,C 180,E1 19541.931,E2 19541.931} C_VEL
LIN {X 0,Y 424.017,Z 1043.207,A -85,B 0,C 180,E1 19540.938,E2 19540.938} C_VEL
LIN {X 0,Y 416.931,Z 1048.169,A -85,B 0,C 180,E1 19538.12,E2 19538.12} C_VEL
LIN {X 0,Y 416.28,Z 1049.288,A -85,B 0,C 180,E1 19537.374,E2 19537.374} C_VEL
LIN {X 0,Y 416,Z 1053.238,A -85,B 0,C 180,E1 19533.859,E2 19533.859} C_VEL
LIN {X 0,Y 415.931,Z 1055.35,A -85,B 0,C 180,E1 19530.826,E2 19530.826} C_VEL
LIN {X 0,Y 415.907,Z 1056.265,A -85,B 0,C 180,E1 19528.071,E2 19528.071} C_VEL
LIN {X 0,Y 415.906,Z 1056.207,A -85,B 0,C 180,E1 19525.311,E2 19525.311} C_VEL
LIN {X 0,Y 415.923,Z 1055.038,A -85,B 0,C 180,E1 19522.263,E2 19522.263} C_VEL
LIN {X 0,Y 416.078,Z 1052.196,A -85,B 0,C 180,E1 19518.776,E2 19518.776} C_VEL
LIN {X 0,Y 416.426,Z 1048.337,A -85,B 0,C 180,E1 19515.681,E2 19515.681} C_VEL
LIN {X 0,Y 417.053,Z 1043.747,A -85,B 0,C 180,E1 19512.849,E2 19512.849} C_VEL
LIN {X 0,Y 418.191,Z 1037.463,A -85,B 0,C 180,E1 19509.715,E2 19509.715} C_VEL
LIN {X 0,Y 420.242,Z 1028.548,A -85,B 0,C 180,E1 19506.141,E2 19506.141} C_VEL
LIN {X 0,Y 422.676,Z 1019.54,A -85,B 0,C 180,E1 19503.139,E2 19503.139} C_VEL
LIN {X 0,Y 425.852,Z 1009.117,A -85,B 0,C 180,E1 19500.148,E2 19500.148} C_VEL
LIN {X 0,Y 430.482,Z 995.129,A -85,B 0,C 180,E1 19496.759,E2 19496.759} C_VEL
LIN {X 0,Y 434.67,Z 983.097,A -85,B 0,C 180,E1 19494.248,E2 19494.248} C_VEL
LIN {X 0,Y 439.802,Z 968.833,A -85,B 0,C 180,E1 19491.635,E2 19491.635} C_VEL
LIN {X 0,Y 446.256,Z 950.945,A -85,B 0,C 180,E1 19488.838,E2 19488.838} C_VEL
LIN {X 0,Y 451.831,Z 935.339,A -85,B 0,C 180,E1 19486.725,E2 19486.725} C_VEL
LIN {X 0,Y 458.143,Z 917.36,A -85,B 0,C 180,E1 19484.594,E2 19484.594} C_VEL
LIN {X 0,Y 465.054,Z 896.44,A -85,B 0,C 180,E1 19482.484,E2 19482.484} C_VEL
LIN {X 0,Y 470.61,Z 878.792,A -85,B 0,C 180,E1 19480.947,E2 19480.947} C_VEL
LIN {X 0,Y 476.711,Z 858.151,A -85,B 0,C 180,E1 19479.384,E2 19479.384} C_VEL
LIN {X 0,Y 482.859,Z 834.982,A -85,B 0,C 180,E1 19477.912,E2 19477.912} C_VEL
LIN {X 0,Y 487.48,Z 815.758,A -85,B 0,C 180,E1 19476.876,E2 19476.876} C_VEL
LIN {X 0,Y 491.695,Z 796.112,A -85,B 0,C 180,E1 19475.967,E2 19475.967} C_VEL
LIN {X 0,Y 496.437,Z 770.557,A -85,B 0,C 180,E1 19474.997,E2 19474.997} C_VEL
LIN {X 0,Y 499.83,Z 747.572,A -85,B 0,C 180,E1 19474.313,E2 19474.313} C_VEL
LIN {X 0,Y 502.467,Z 725.352,A -85,B 0,C 180,E1 19473.799,E2 19473.799} C_VEL
LIN {X 0,Y 504.772,Z 695.148,A -85,B 0,C 180,E1 19473.274,E2 19473.274} C_VEL
LIN {X 0,Y 517.706,Z 465.936,A -85,B 0,C 180,E1 19469.723,E2 19469.723} C_VEL
LIN {X 0,Y 520.492,Z 417.274,A -85,B 0,C 180,E1 19468.954,E2 19468.954} C_VEL
LIN {X 0,Y 509.665,Z 399.94,A -85,B 0,C 180,E1 19466.32,E2 19466.32} C_VEL
LIN {X 0,Y 502.31,Z 389.586,A -85,B 0,C 180,E1 19464.365,E2 19464.365} C_VEL
LIN {X 0,Y 494.658,Z 379.23,A -85,B 0,C 180,E1 19462.116,E2 19462.116} C_VEL
LIN {X 0,Y 488.219,Z 370.764,A -85,B 0,C 180,E1 19460,E2 19460} C_VEL
LIN {X 0,Y 483.28,Z 364.641,A -85,B 0,C 180,E1 19458.205,E2 19458.205} C_VEL
LIN {X 0,Y 479.18,Z 359.475,A -85,B 0,C 180,E1 19456.549,E2 19456.549} C_VEL
LIN {X 0,Y 475.425,Z 354.885,A -85,B 0,C 180,E1 19454.868,E2 19454.868} C_VEL
LIN {X 0,Y 474.199,Z 353.528,A -85,B 0,C 180,E1 19454.283,E2 19454.283} C_VEL
LIN {X 0,Y 470.913,Z 349.704,A -85,B 0,C 180,E1 19452.57,E2 19452.57} C_VEL
LIN {X 0,Y 469.811,Z 347.975,A -85,B 0,C 180,E1 19451.914,E2 19451.914} C_VEL
LIN {X 0,Y 466.272,Z 344.585,A -85,B 0,C 180,E1 19449.691,E2 19449.691} C_VEL
LIN {X 0,Y 464.848,Z 341.91,A -85,B 0,C 180,E1 19448.535,E2 19448.535} C_VEL
LIN {X 0,Y 461.169,Z 338.868,A -85,B 0,C 180,E1 19445.1,E2 19445.1} C_VEL
LIN {X 0,Y 459.674,Z 335.876,A -85,B 0,C 180,E1 19442.618,E2 19442.618} C_VEL
LIN {X 0,Y 458.604,Z 335.14,A -85,B 0,C 180,E1 19438.751,E2 19438.751} C_VEL
LIN {X 0,Y 459.728,Z 335.887,A -85,B 0,C 180,E1 19434.383,E2 19434.383} C_VEL
LIN {X 0,Y 462.733,Z 340.654,A -85,B 0,C 180,E1 19430.297,E2 19430.297} C_VEL
LIN {X 0,Y 465.04,Z 342.17,A -85,B 0,C 180,E1 19428.402,E2 19428.402} C_VEL
LIN {X 0,Y 467.379,Z 345.916,A -85,B 0,C 180,E1 19426.641,E2 19426.641} C_VEL
LIN {X 0,Y 470.28,Z 348.613,A -85,B 0,C 180,E1 19424.903,E2 19424.903} C_VEL
LIN {X 0,Y 473.306,Z 352.752,A -85,B 0,C 180,E1 19423.24,E2 19423.24} C_VEL
LIN {X 0,Y 475.396,Z 354.768,A -85,B 0,C 180,E1 19422.243,E2 19422.243} C_VEL
LIN {X 0,Y 479.152,Z 359.438,A -85,B 0,C 180,E1 19420.558,E2 19420.558} C_VEL
LIN {X 0,Y 485.057,Z 366.904,A -85,B 0,C 180,E1 19418.22,E2 19418.22} C_VEL
LIN {X 0,Y 489.806,Z 373.018,A -85,B 0,C 180,E1 19416.542,E2 19416.542} C_VEL
LIN {X 0,Y 495.296,Z 380.779,A -85,B 0,C 180,E1 19414.756,E2 19414.756} C_VEL
LIN {X 0,Y 503.781,Z 393.028,A -85,B 0,C 180,E1 19412.284,E2 19412.284} C_VEL
LIN {X 0,Y 514.334,Z 409.622,A -85,B 0,C 180,E1 19409.542,E2 19409.542} C_VEL
LIN {X 0,Y 520.52,Z 420.326,A -85,B 0,C 180,E1 19408.06,E2 19408.06} C_VEL
LIN {X 0,Y 507.691,Z 644.053,A -85,B 0,C 180,E1 19404.593,E2 19404.593} C_VEL
LIN {X 0,Y 503.276,Z 720.374,A -85,B 0,C 180,E1 19403.389,E2 19403.389} C_VEL
LIN {X 0,Y 500.294,Z 748.349,A -85,B 0,C 180,E1 19402.803,E2 19402.803} C_VEL
LIN {X 0,Y 497.248,Z 769.296,A -85,B 0,C 180,E1 19402.227,E2 19402.227} C_VEL
LIN {X 0,Y 493.538,Z 790.697,A -85,B 0,C 180,E1 19401.497,E2 19401.497} C_VEL
LIN {X 0,Y 488.136,Z 817.082,A -85,B 0,C 180,E1 19400.371,E2 19400.371} C_VEL
LIN {X 0,Y 483.045,Z 838.477,A -85,B 0,C 180,E1 19399.254,E2 19399.254} C_VEL
LIN {X 0,Y 477.683,Z 858.992,A -85,B 0,C 180,E1 19397.995,E2 19397.995} C_VEL
LIN {X 0,Y 470.719,Z 883.057,A -85,B 0,C 180,E1 19396.238,E2 19396.238} C_VEL
LIN {X 0,Y 465.019,Z 901.276,A -85,B 0,C 180,E1 19394.677,E2 19394.677} C_VEL
LIN {X 0,Y 458.765,Z 920.362,A -85,B 0,C 180,E1 19392.801,E2 19392.801} C_VEL
LIN {X 0,Y 451.967,Z 940.087,A -85,B 0,C 180,E1 19390.529,E2 19390.529} C_VEL
LIN {X 0,Y 446.548,Z 955.404,A -85,B 0,C 180,E1 19388.498,E2 19388.498} C_VEL
LIN {X 0,Y 441.136,Z 970.637,A -85,B 0,C 180,E1 19386.204,E2 19386.204} C_VEL
LIN {X 0,Y 434.985,Z 987.996,A -85,B 0,C 180,E1 19383.167,E2 19383.167} C_VEL
LIN {X 0,Y 430.573,Z 1000.761,A -85,B 0,C 180,E1 19380.568,E2 19380.568} C_VEL
LIN {X 0,Y 426.692,Z 1012.689,A -85,B 0,C 180,E1 19377.796,E2 19377.796} C_VEL
LIN {X 0,Y 422.822,Z 1025.511,A -85,B 0,C 180,E1 19374.297,E2 19374.297} C_VEL
LIN {X 0,Y 420.354,Z 1034.675,A -85,B 0,C 180,E1 19371.342,E2 19371.342} C_VEL
LIN {X 0,Y 418.486,Z 1042.886,A -85,B 0,C 180,E1 19368.24,E2 19368.24} C_VEL
LIN {X 0,Y 417.069,Z 1050.741,A -85,B 0,C 180,E1 19364.58,E2 19364.58} C_VEL
LIN {X 0,Y 416.383,Z 1055.866,A -85,B 0,C 180,E1 19361.546,E2 19361.546} C_VEL
LIN {X 0,Y 416.061,Z 1059.586,A -85,B 0,C 180,E1 19358.708,E2 19358.708} C_VEL
LIN {X 0,Y 415.928,Z 1062.333,A -85,B 0,C 180,E1 19355.795,E2 19355.795} C_VEL
LIN {X 0,Y 415.909,Z 1064.176,A -85,B 0,C 180,E1 19352.342,E2 19352.342} C_VEL
LIN {X 0,Y 415.909,Z 1064.427,A -85,B 0,C 180,E1 19349.311,E2 19349.311} C_VEL
LIN {X 0,Y 415.911,Z 1063.64,A -85,B 0,C 180,E1 19346.554,E2 19346.554} C_VEL
LIN {X 0,Y 415.947,Z 1061.857,A -85,B 0,C 180,E1 19343.79,E2 19343.79} C_VEL
LIN {X 0,Y 416.076,Z 1059.052,A -85,B 0,C 180,E1 19341.003,E2 19341.003} C_VEL
LIN {X 0,Y 416.515,Z 1054.463,A -85,B 0,C 180,E1 19337.702,E2 19337.702} C_VEL
LIN {X 0,Y 417.448,Z 1047.752,A -85,B 0,C 180,E1 19334.154,E2 19334.154} C_VEL
LIN {X 0,Y 418.728,Z 1040.839,A -85,B 0,C 180,E1 19331.194,E2 19331.194} C_VEL
LIN {X 0,Y 420.701,Z 1032.24,A -85,B 0,C 180,E1 19328.09,E2 19328.09} C_VEL
LIN {X 0,Y 423.698,Z 1020.842,A -85,B 0,C 180,E1 19324.669,E2 19324.669} C_VEL
LIN {X 0,Y 426.862,Z 1010.088,A -85,B 0,C 180,E1 19321.912,E2 19321.912} C_VEL
LIN {X 0,Y 430.98,Z 997.062,A -85,B 0,C 180,E1 19319,E2 19319} C_VEL
LIN {X 0,Y 436.179,Z 981.232,A -85,B 0,C 180,E1 19315.99,E2 19315.99} C_VEL
LIN {X 0,Y 440.821,Z 967.399,A -85,B 0,C 180,E1 19313.7,E2 19313.7} C_VEL
LIN {X 0,Y 446.766,Z 949.879,A -85,B 0,C 180,E1 19311.155,E2 19311.155} C_VEL
LIN {X 0,Y 452.963,Z 931.011,A -85,B 0,C 180,E1 19308.828,E2 19308.828} C_VEL
LIN {X 0,Y 458.331,Z 914.244,A -85,B 0,C 180,E1 19307.02,E2 19307.02} C_VEL
LIN {X 0,Y 464.823,Z 893.252,A -85,B 0,C 180,E1 19305.05,E2 19305.05} C_VEL
LIN {X 0,Y 470.693,Z 872.532,A -85,B 0,C 180,E1 19303.406,E2 19303.406} C_VEL
LIN {X 0,Y 475.71,Z 853.581,A -85,B 0,C 180,E1 19302.101,E2 19302.101} C_VEL
LIN {X 0,Y 481.224,Z 831.025,A -85,B 0,C 180,E1 19300.769,E2 19300.769} C_VEL
LIN {X 0,Y 486.32,Z 806.858,A -85,B 0,C 180,E1 19299.596,E2 19299.596} C_VEL
LIN {X 0,Y 490.186,Z 785.921,A -85,B 0,C 180,E1 19298.752,E2 19298.752} C_VEL
LIN {X 0,Y 494.214,Z 760.418,A -85,B 0,C 180,E1 19297.919,E2 19297.919} C_VEL
LIN {X 0,Y 497.231,Z 735.211,A -85,B 0,C 180,E1 19297.309,E2 19297.309} C_VEL
LIN {X 0,Y 499.129,Z 712.651,A -85,B 0,C 180,E1 19296.889,E2 19296.889} C_VEL
LIN {X 0,Y 511.336,Z 479.982,A -85,B 0,C 180,E1 19293.288,E2 19293.288} C_VEL
LIN {X 0,Y 514.637,Z 417.101,A -85,B 0,C 180,E1 19292.297,E2 19292.297} C_VEL
LIN {X 0,Y 505.128,Z 401.049,A -85,B 0,C 180,E1 19290.218,E2 19290.218} C_VEL
LIN {X 0,Y 494.755,Z 384.655,A -85,B 0,C 180,E1 19287.732,E2 19287.732} C_VEL
LIN {X 0,Y 483.748,Z 368.514,A -85,B 0,C 180,E1 19284.776,E2 19284.776} C_VEL
LIN {X 0,Y 478.015,Z 361.321,A -85,B 0,C 180,E1 19283.092,E2 19283.092} C_VEL
LIN {X 0,Y 473.936,Z 356.166,A -85,B 0,C 180,E1 19281.797,E2 19281.797} C_VEL
LIN {X 0,Y 470.069,Z 351.3,A -85,B 0,C 180,E1 19280.482,E2 19280.482} C_VEL
LIN {X 0,Y 466.197,Z 346.371,A -85,B 0,C 180,E1 19279.059,E2 19279.059} C_VEL
LIN {X 0,Y 462.156,Z 341.864,A -85,B 0,C 180,E1 19277.469,E2 19277.469} C_VEL
LIN {X 0,Y 460.842,Z 340.086,A -85,B 0,C 180,E1 19276.902,E2 19276.902} C_VEL
LIN {X 0,Y 457.469,Z 336.535,A -85,B 0,C 180,E1 19275.4,E2 19275.4} C_VEL
LIN {X 0,Y 455.905,Z 334.136,A -85,B 0,C 180,E1 19274.609,E2 19274.609} C_VEL
LIN {X 0,Y 452.357,Z 330.872,A -85,B 0,C 180,E1 19272.77,E2 19272.77} C_VEL
LIN {X 0,Y 450.579,Z 327.875,A -85,B 0,C 180,E1 19271.651,E2 19271.651} C_VEL
LIN {X 0,Y 447.134,Z 325.24,A -85,B 0,C 180,E1 19269.395,E2 19269.395} C_VEL
LIN {X 0,Y 445.273,Z 321.761,A -85,B 0,C 180,E1 19267.743,E2 19267.743} C_VEL
LIN {X 0,Y 440.071,Z 317.106,A -85,B 0,C 180,E1 19259.609,E2 19259.609} C_VEL
LIN {X 0,Y 440.047,Z 317.088,A -85,B 0,C 180,E1 19257.395,E2 19257.395} C_VEL
LIN {X 0,Y 441.198,Z 318.961,A -85,B 0,C 180,E1 19253.755,E2 19253.755} C_VEL
LIN {X 0,Y 445.292,Z 321.773,A -85,B 0,C 180,E1 19249.062,E2 19249.062} C_VEL
LIN {X 0,Y 447.076,Z 325.165,A -85,B 0,C 180,E1 19247.47,E2 19247.47} C_VEL
LIN {X 0,Y 450.909,Z 328.319,A -85,B 0,C 180,E1 19244.963,E2 19244.963} C_VEL
LIN {X 0,Y 453.39,Z 332.111,A -85,B 0,C 180,E1 19243.471,E2 19243.471} C_VEL
LIN {X 0,Y 456.403,Z 334.734,A -85,B 0,C 180,E1 19241.964,E2 19241.964} C_VEL
LIN {X 0,Y 459.359,Z 338.812,A -85,B 0,C 180,E1 19240.547,E2 19240.547} C_VEL
LIN {X 0,Y 461.545,Z 340.899,A -85,B 0,C 180,E1 19239.62,E2 19239.62} C_VEL
LIN {X 0,Y 464.951,Z 345.235,A -85,B 0,C 180,E1 19238.225,E2 19238.225} C_VEL
LIN {X 0,Y 466.74,Z 347.166,A -85,B 0,C 180,E1 19237.551,E2 19237.551} C_VEL
LIN {X 0,Y 471.595,Z 353.137,A -85,B 0,C 180,E1 19235.812,E2 19235.812} C_VEL
LIN {X 0,Y 476.265,Z 359.057,A -85,B 0,C 180,E1 19234.274,E2 19234.274} C_VEL
LIN {X 0,Y 481.317,Z 365.538,A -85,B 0,C 180,E1 19232.737,E2 19232.737} C_VEL
LIN {X 0,Y 487.572,Z 373.547,A -85,B 0,C 180,E1 19230.987,E2 19230.987} C_VEL
LIN {X 0,Y 498.121,Z 388.172,A -85,B 0,C 180,E1 19228.303,E2 19228.303} C_VEL
LIN {X 0,Y 505.208,Z 398.746,A -85,B 0,C 180,E1 19226.652,E2 19226.652} C_VEL
LIN {X 0,Y 514.776,Z 414.629,A -85,B 0,C 180,E1 19224.566,E2 19224.566} C_VEL
LIN {X 0,Y 503.842,Z 620.182,A -85,B 0,C 180,E1 19221.384,E2 19221.384} C_VEL
LIN {X 0,Y 498.83,Z 713.848,A -85,B 0,C 180,E1 19219.917,E2 19219.917} C_VEL
LIN {X 0,Y 496.03,Z 742.069,A -85,B 0,C 180,E1 19219.321,E2 19219.321} C_VEL
LIN {X 0,Y 493.16,Z 763.311,A -85,B 0,C 180,E1 19218.721,E2 19218.721} C_VEL
LIN {X 0,Y 489.775,Z 784.141,A -85,B 0,C 180,E1 19217.997,E2 19217.997} C_VEL
LIN {X 0,Y 484.848,Z 809.911,A -85,B 0,C 180,E1 19216.89,E2 19216.89} C_VEL
LIN {X 0,Y 480.051,Z 831.307,A -85,B 0,C 180,E1 19215.767,E2 19215.767} C_VEL
LIN {X 0,Y 475.207,Z 850.904,A -85,B 0,C 180,E1 19214.565,E2 19214.565} C_VEL
LIN {X 0,Y 468.859,Z 874.408,A -85,B 0,C 180,E1 19212.867,E2 19212.867} C_VEL
LIN {X 0,Y 463.045,Z 894.014,A -85,B 0,C 180,E1 19211.194,E2 19211.194} C_VEL
LIN {X 0,Y 457.416,Z 912.109,A -85,B 0,C 180,E1 19209.421,E2 19209.421} C_VEL
LIN {X 0,Y 450.454,Z 933.431,A -85,B 0,C 180,E1 19206.981,E2 19206.981} C_VEL
LIN {X 0,Y 445.247,Z 948.831,A -85,B 0,C 180,E1 19204.935,E2 19204.935} C_VEL
LIN {X 0,Y 440.236,Z 963.538,A -85,B 0,C 180,E1 19202.721,E2 19202.721} C_VEL
LIN {X 0,Y 434.297,Z 981.007,A -85,B 0,C 180,E1 19199.669,E2 19199.669} C_VEL
LIN {X 0,Y 430.058,Z 993.789,A -85,B 0,C 180,E1 19197.066,E2 19197.066} C_VEL
LIN {X 0,Y 426.059,Z 1006.499,A -85,B 0,C 180,E1 19194.101,E2 19194.101} C_VEL
LIN {X 0,Y 422.563,Z 1018.452,A -85,B 0,C 180,E1 19190.789,E2 19190.789} C_VEL
LIN {X 0,Y 420.321,Z 1027.019,A -85,B 0,C 180,E1 19188.014,E2 19188.014} C_VEL
LIN {X 0,Y 418.509,Z 1035.099,A -85,B 0,C 180,E1 19184.953,E2 19184.953} C_VEL
LIN {X 0,Y 417.115,Z 1042.835,A -85,B 0,C 180,E1 19181.336,E2 19181.336} C_VEL
LIN {X 0,Y 416.442,Z 1047.753,A -85,B 0,C 180,E1 19178.416,E2 19178.416} C_VEL
LIN {X 0,Y 416.28,Z 1049.288,A -85,B 0,C 180,E1 19177.374,E2 19177.374} C_VEL
LIN {X 0,Y 415.158,Z 1050.718,A -85,B 0,C 180,E1 19176.334,E2 19176.334} C_VEL
LIN {X 0,Y 408.605,Z 1053.721,A -85,B 0,C 180,E1 19173.462,E2 19173.462} C_VEL
LIN {X 0,Y 407.945,Z 1054.407,A -85,B 0,C 180,E1 19172.611,E2 19172.611} C_VEL
LIN {X 0,Y 407.913,Z 1056.169,A -85,B 0,C 180,E1 19169.157,E2 19169.157} C_VEL
LIN {X 0,Y 407.906,Z 1056.391,A -85,B 0,C 180,E1 19165.924,E2 19165.924} C_VEL
LIN {X 0,Y 407.934,Z 1055.556,A -85,B 0,C 180,E1 19163.075,E2 19163.075} C_VEL
LIN {X 0,Y 407.998,Z 1053.763,A -85,B 0,C 180,E1 19160.265,E2 19160.265} C_VEL
LIN {X 0,Y 408.213,Z 1050.796,A -85,B 0,C 180,E1 19157.265,E2 19157.265} C_VEL
LIN {X 0,Y 408.884,Z 1045.535,A -85,B 0,C 180,E1 19153.521,E2 19153.521} C_VEL
LIN {X 0,Y 409.956,Z 1039.517,A -85,B 0,C 180,E1 19150.299,E2 19150.299} C_VEL
LIN {X 0,Y 411.425,Z 1033.013,A -85,B 0,C 180,E1 19147.419,E2 19147.419} C_VEL
LIN {X 0,Y 413.994,Z 1023.632,A -85,B 0,C 180,E1 19143.924,E2 19143.924} C_VEL
LIN {X 0,Y 417.346,Z 1012.68,A -85,B 0,C 180,E1 19140.584,E2 19140.584} C_VEL
LIN {X 0,Y 420.839,Z 1002.3,A -85,B 0,C 180,E1 19137.845,E2 19137.845} C_VEL
LIN {X 0,Y 425.824,Z 988.631,A -85,B 0,C 180,E1 19134.715,E2 19134.715} C_VEL
LIN {X 0,Y 431.428,Z 973.368,A -85,B 0,C 180,E1 19131.771,E2 19131.771} C_VEL
LIN {X 0,Y 436.652,Z 959.488,A -85,B 0,C 180,E1 19129.434,E2 19129.434} C_VEL
LIN {X 0,Y 443.6,Z 941.053,A -85,B 0,C 180,E1 19126.747,E2 19126.747} C_VEL
LIN {X 0,Y 449.793,Z 924.014,A -85,B 0,C 180,E1 19124.626,E2 19124.626} C_VEL
LIN {X 0,Y 455.697,Z 907.279,A -85,B 0,C 180,E1 19122.801,E2 19122.801} C_VEL
LIN {X 0,Y 462.893,Z 885.922,A -85,B 0,C 180,E1 19120.79,E2 19120.79} C_VEL
LIN {X 0,Y 469.04,Z 866.023,A -85,B 0,C 180,E1 19119.204,E2 19119.204} C_VEL
LIN {X 0,Y 474.238,Z 847.932,A -85,B 0,C 180,E1 19117.95,E2 19117.95} C_VEL
LIN {X 0,Y 480.203,Z 825.407,A -85,B 0,C 180,E1 19116.612,E2 19116.612} C_VEL
LIN {X 0,Y 485.617,Z 801.704,A -85,B 0,C 180,E1 19115.452,E2 19115.452} C_VEL
LIN {X 0,Y 489.828,Z 780.544,A -85,B 0,C 180,E1 19114.593,E2 19114.593} C_VEL
LIN {X 0,Y 494.069,Z 755.599,A -85,B 0,C 180,E1 19113.771,E2 19113.771} C_VEL
LIN {X 0,Y 497.374,Z 729.803,A -85,B 0,C 180,E1 19113.14,E2 19113.14} C_VEL
LIN {X 0,Y 499.408,Z 707.547,A -85,B 0,C 180,E1 19112.723,E2 19112.723} C_VEL
LIN {X 0,Y 513.043,Z 474.856,A -85,B 0,C 180,E1 19109.098,E2 19109.098} C_VEL
LIN {X 0,Y 516.132,Z 421.516,A -85,B 0,C 180,E1 19108.241,E2 19108.241} C_VEL
LIN {X 0,Y 506.252,Z 405.616,A -85,B 0,C 180,E1 19105.755,E2 19105.755} C_VEL
LIN {X 0,Y 498.961,Z 395.299,A -85,B 0,C 180,E1 19103.753,E2 19103.753} C_VEL
LIN {X 0,Y 491.935,Z 385.669,A -85,B 0,C 180,E1 19101.617,E2 19101.617} C_VEL
LIN {X 0,Y 485.631,Z 377.428,A -85,B 0,C 180,E1 19099.485,E2 19099.485} C_VEL
LIN {X 0,Y 481.41,Z 372.019,A -85,B 0,C 180,E1 19097.903,E2 19097.903} C_VEL
LIN {X 0,Y 477.519,Z 367.03,A -85,B 0,C 180,E1 19096.295,E2 19096.295} C_VEL
LIN {X 0,Y 473.712,Z 362.236,A -85,B 0,C 180,E1 19094.547,E2 19094.547} C_VEL
LIN {X 0,Y 469.505,Z 357.406,A -85,B 0,C 180,E1 19092.359,E2 19092.359} C_VEL
LIN {X 0,Y 468.418,Z 355.716,A -85,B 0,C 180,E1 19091.7,E2 19091.7} C_VEL
LIN {X 0,Y 464.877,Z 352.143,A -85,B 0,C 180,E1 19089.408,E2 19089.408} C_VEL
LIN {X 0,Y 463.555,Z 349.71,A -85,B 0,C 180,E1 19088.31,E2 19088.31} C_VEL
LIN {X 0,Y 460.091,Z 346.745,A -85,B 0,C 180,E1 19084.987,E2 19084.987} C_VEL
LIN {X 0,Y 458.635,Z 343.769,A -85,B 0,C 180,E1 19082.499,E2 19082.499} C_VEL
LIN {X 0,Y 457.625,Z 343.081,A -85,B 0,C 180,E1 19078.498,E2 19078.498} C_VEL
LIN {X 0,Y 458.754,Z 343.847,A -85,B 0,C 180,E1 19074.371,E2 19074.371} C_VEL
LIN {X 0,Y 461.506,Z 348.431,A -85,B 0,C 180,E1 19070.522,E2 19070.522} C_VEL
LIN {X 0,Y 463.827,Z 350.05,A -85,B 0,C 180,E1 19068.561,E2 19068.561} C_VEL
LIN {X 0,Y 466.228,Z 353.82,A -85,B 0,C 180,E1 19066.734,E2 19066.734} C_VEL
LIN {X 0,Y 468.891,Z 356.354,A -85,B 0,C 180,E1 19065.11,E2 19065.11} C_VEL
LIN {X 0,Y 471.992,Z 360.561,A -85,B 0,C 180,E1 19063.382,E2 19063.382} C_VEL
LIN {X 0,Y 473.81,Z 362.333,A -85,B 0,C 180,E1 19062.499,E2 19062.499} C_VEL
LIN {X 0,Y 477.57,Z 367.065,A -85,B 0,C 180,E1 19060.779,E2 19060.779} C_VEL
LIN {X 0,Y 483.396,Z 374.604,A -85,B 0,C 180,E1 19058.428,E2 19058.428} C_VEL
LIN {X 0,Y 488.012,Z 380.615,A -85,B 0,C 180,E1 19056.77,E2 19056.77} C_VEL
LIN {X 0,Y 493.347,Z 388.317,A -85,B 0,C 180,E1 19055.002,E2 19055.002} C_VEL
LIN {X 0,Y 501.606,Z 400.47,A -85,B 0,C 180,E1 19052.55,E2 19052.55} C_VEL
LIN {X 0,Y 511.862,Z 416.905,A -85,B 0,C 180,E1 19049.833,E2 19049.833} C_VEL
LIN {X 0,Y 516.206,Z 424.585,A -85,B 0,C 180,E1 19048.761,E2 19048.761} C_VEL
LIN {X 0,Y 503.018,Z 647.712,A -85,B 0,C 180,E1 19045.292,E2 19045.292} C_VEL
LIN {X 0,Y 498.666,Z 720.448,A -85,B 0,C 180,E1 19044.14,E2 19044.14} C_VEL
LIN {X 0,Y 495.607,Z 748.378,A -85,B 0,C 180,E1 19043.554,E2 19043.554} C_VEL
LIN {X 0,Y 492.479,Z 769.305,A -85,B 0,C 180,E1 19042.979,E2 19042.979} C_VEL
LIN {X 0,Y 488.59,Z 791.151,A -85,B 0,C 180,E1 19042.232,E2 19042.232} C_VEL
LIN {X 0,Y 483.041,Z 817.412,A -85,B 0,C 180,E1 19041.106,E2 19041.106} C_VEL
LIN {X 0,Y 477.976,Z 838.13,A -85,B 0,C 180,E1 19040.023,E2 19040.023} C_VEL
LIN {X 0,Y 472.542,Z 858.344,A -85,B 0,C 180,E1 19038.784,E2 19038.784} C_VEL
LIN {X 0,Y 465.35,Z 882.51,A -85,B 0,C 180,E1 19037.023,E2 19037.023} C_VEL
LIN {X 0,Y 459.459,Z 900.771,A -85,B 0,C 180,E1 19035.456,E2 19035.456} C_VEL
LIN {X 0,Y 453.214,Z 919.184,A -85,B 0,C 180,E1 19033.644,E2 19033.644} C_VEL
LIN {X 0,Y 445.816,Z 939.921,A -85,B 0,C 180,E1 19031.253,E2 19031.253} C_VEL
LIN {X 0,Y 440.089,Z 955.487,A -85,B 0,C 180,E1 19029.17,E2 19029.17} C_VEL
LIN {X 0,Y 434.584,Z 970.359,A -85,B 0,C 180,E1 19026.906,E2 19026.906} C_VEL
LIN {X 0,Y 428.049,Z 988.035,A -85,B 0,C 180,E1 19023.776,E2 19023.776} C_VEL
LIN {X 0,Y 423.425,Z 1000.788,A -85,B 0,C 180,E1 19021.141,E2 19021.141} C_VEL
LIN {X 0,Y 419.169,Z 1013.276,A -85,B 0,C 180,E1 19018.184,E2 19018.184} C_VEL
LIN {X 0,Y 415.264,Z 1025.505,A -85,B 0,C 180,E1 19014.769,E2 19014.769} C_VEL
LIN {X 0,Y 412.659,Z 1034.659,A -85,B 0,C 180,E1 19011.76,E2 19011.76} C_VEL
LIN {X 0,Y 410.671,Z 1042.861,A -85,B 0,C 180,E1 19008.6,E2 19008.6} C_VEL
LIN {X 0,Y 409.157,Z 1050.699,A -85,B 0,C 180,E1 19004.868,E2 19004.868} C_VEL
LIN {X 0,Y 408.439,Z 1055.681,A -85,B 0,C 180,E1 19001.867,E2 19001.867} C_VEL
LIN {X 0,Y 408.082,Z 1059.369,A -85,B 0,C 180,E1 18999.022,E2 18999.022} C_VEL
LIN {X 0,Y 407.946,Z 1062.042,A -85,B 0,C 180,E1 18996.191,E2 18996.191} C_VEL
LIN {X 0,Y 407.914,Z 1063.991,A -85,B 0,C 180,E1 18992.81,E2 18992.81} C_VEL
LIN {X 0,Y 407.909,Z 1064.369,A -85,B 0,C 180,E1 18989.438,E2 18989.438} C_VEL
LIN {X 0,Y 407.911,Z 1063.553,A -85,B 0,C 180,E1 18986.487,E2 18986.487} C_VEL
LIN {X 0,Y 407.953,Z 1061.763,A -85,B 0,C 180,E1 18983.668,E2 18983.668} C_VEL
LIN {X 0,Y 408.091,Z 1058.962,A -85,B 0,C 180,E1 18980.836,E2 18980.836} C_VEL
LIN {X 0,Y 408.567,Z 1054.295,A -85,B 0,C 180,E1 18977.42,E2 18977.42} C_VEL
LIN {X 0,Y 409.561,Z 1047.627,A -85,B 0,C 180,E1 18973.84,E2 18973.84} C_VEL
LIN {X 0,Y 410.927,Z 1040.704,A -85,B 0,C 180,E1 18970.823,E2 18970.823} C_VEL
LIN {X 0,Y 413.137,Z 1031.685,A -85,B 0,C 180,E1 18967.518,E2 18967.518} C_VEL
LIN {X 0,Y 416.3,Z 1020.312,A -85,B 0,C 180,E1 18964.079,E2 18964.079} C_VEL
LIN {X 0,Y 419.658,Z 1009.442,A -85,B 0,C 180,E1 18961.26,E2 18961.26} C_VEL
LIN {X 0,Y 424.312,Z 995.57,A -85,B 0,C 180,E1 18958.14,E2 18958.14} C_VEL
LIN {X 0,Y 429.534,Z 980.237,A -85,B 0,C 180,E1 18955.228,E2 18955.228} C_VEL
LIN {X 0,Y 434.406,Z 966.315,A -85,B 0,C 180,E1 18952.911,E2 18952.911} C_VEL
LIN {X 0,Y 440.903,Z 947.859,A -85,B 0,C 180,E1 18950.244,E2 18950.244} C_VEL
LIN {X 0,Y 446.881,Z 930.31,A -85,B 0,C 180,E1 18948.078,E2 18948.078} C_VEL
LIN {X 0,Y 452.506,Z 913.331,A -85,B 0,C 180,E1 18946.241,E2 18946.241} C_VEL
LIN {X 0,Y 459.468,Z 891.318,A -85,B 0,C 180,E1 18944.189,E2 18944.189} C_VEL
LIN {X 0,Y 465.334,Z 871.212,A -85,B 0,C 180,E1 18942.599,E2 18942.599} C_VEL
LIN {X 0,Y 470.37,Z 852.722,A -85,B 0,C 180,E1 18941.33,E2 18941.33} C_VEL
LIN {X 0,Y 476.179,Z 829.499,A -85,B 0,C 180,E1 18939.966,E2 18939.966} C_VEL
LIN {X 0,Y 481.122,Z 806.524,A -85,B 0,C 180,E1 18938.857,E2 18938.857} C_VEL
LIN {X 0,Y 484.959,Z 786.27,A -85,B 0,C 180,E1 18938.038,E2 18938.038} C_VEL
LIN {X 0,Y 489.081,Z 761.004,A -85,B 0,C 180,E1 18937.207,E2 18937.207} C_VEL
LIN {X 0,Y 492.241,Z 735.331,A -85,B 0,C 180,E1 18936.583,E2 18936.583} C_VEL
LIN {X 0,Y 494.189,Z 712.836,A -85,B 0,C 180,E1 18936.162,E2 18936.162} C_VEL
LIN {X 0,Y 506.786,Z 480.48,A -85,B 0,C 180,E1 18932.549,E2 18932.549} C_VEL
LIN {X 0,Y 509.976,Z 421.093,A -85,B 0,C 180,E1 18931.604,E2 18931.604} C_VEL
LIN {X 0,Y 501.531,Z 406.746,A -85,B 0,C 180,E1 18929.698,E2 18929.698} C_VEL
LIN {X 0,Y 491.863,Z 391.229,A -85,B 0,C 180,E1 18927.318,E2 18927.318} C_VEL
LIN {X 0,Y 481.225,Z 375.382,A -85,B 0,C 180,E1 18924.391,E2 18924.391} C_VEL
LIN {X 0,Y 472.617,Z 364.268,A -85,B 0,C 180,E1 18921.73,E2 18921.73} C_VEL
LIN {X 0,Y 467.775,Z 358.339,A -85,B 0,C 180,E1 18920.064,E2 18920.064} C_VEL
LIN {X 0,Y 463.594,Z 353.111,A -85,B 0,C 180,E1 18918.485,E2 18918.485} C_VEL
LIN {X 0,Y 459.858,Z 348.462,A -85,B 0,C 180,E1 18916.94,E2 18916.94} C_VEL
LIN {X 0,Y 455.612,Z 343.704,A -85,B 0,C 180,E1 18915.009,E2 18915.009} C_VEL
LIN {X 0,Y 454.435,Z 341.857,A -85,B 0,C 180,E1 18914.397,E2 18914.397} C_VEL
LIN {X 0,Y 450.841,Z 338.41,A -85,B 0,C 180,E1 18912.488,E2 18912.488} C_VEL
LIN {X 0,Y 449.19,Z 335.65,A -85,B 0,C 180,E1 18911.427,E2 18911.427} C_VEL
LIN {X 0,Y 445.745,Z 332.834,A -85,B 0,C 180,E1 18909.099,E2 18909.099} C_VEL
LIN {X 0,Y 443.873,Z 329.354,A -85,B 0,C 180,E1 18907.377,E2 18907.377} C_VEL
LIN {X 0,Y 439.079,Z 325.022,A -85,B 0,C 180,E1 18899.478,E2 18899.478} C_VEL
LIN {X 0,Y 439.087,Z 325.062,A -85,B 0,C 180,E1 18897.259,E2 18897.259} C_VEL
LIN {X 0,Y 444.04,Z 329.497,A -85,B 0,C 180,E1 18889.294,E2 18889.294} C_VEL
LIN {X 0,Y 445.777,Z 332.869,A -85,B 0,C 180,E1 18887.697,E2 18887.697} C_VEL
LIN {X 0,Y 449.526,Z 336.089,A -85,B 0,C 180,E1 18885.179,E2 18885.179} C_VEL
LIN {X 0,Y 452.086,Z 339.925,A -85,B 0,C 180,E1 18883.621,E2 18883.621} C_VEL
LIN {X 0,Y 454.856,Z 342.398,A -85,B 0,C 180,E1 18882.208,E2 18882.208} C_VEL
LIN {X 0,Y 457.995,Z 346.641,A -85,B 0,C 180,E1 18880.685,E2 18880.685} C_VEL
LIN {X 0,Y 459.937,Z 348.617,A -85,B 0,C 180,E1 18879.844,E2 18879.844} C_VEL
LIN {X 0,Y 463.542,Z 353.077,A -85,B 0,C 180,E1 18878.355,E2 18878.355} C_VEL
LIN {X 0,Y 465.294,Z 355.223,A -85,B 0,C 180,E1 18877.677,E2 18877.677} C_VEL
LIN {X 0,Y 469.708,Z 360.645,A -85,B 0,C 180,E1 18876.076,E2 18876.076} C_VEL
LIN {X 0,Y 474.231,Z 366.457,A -85,B 0,C 180,E1 18874.558,E2 18874.558} C_VEL
LIN {X 0,Y 481.793,Z 376.14,A -85,B 0,C 180,E1 18872.264,E2 18872.264} C_VEL
LIN {X 0,Y 492.002,Z 390.149,A -85,B 0,C 180,E1 18869.506,E2 18869.506} C_VEL
LIN {X 0,Y 500.639,Z 402.856,A -85,B 0,C 180,E1 18867.401,E2 18867.401} C_VEL
LIN {X 0,Y 510.141,Z 418.674,A -85,B 0,C 180,E1 18865.253,E2 18865.253} C_VEL
LIN {X 0,Y 498.859,Z 624.228,A -85,B 0,C 180,E1 18862.058,E2 18862.058} C_VEL
LIN {X 0,Y 493.893,Z 713.997,A -85,B 0,C 180,E1 18860.645,E2 18860.645} C_VEL
LIN {X 0,Y 491.015,Z 742.255,A -85,B 0,C 180,E1 18860.046,E2 18860.046} C_VEL
LIN {X 0,Y 488.084,Z 763.373,A -85,B 0,C 180,E1 18859.45,E2 18859.45} C_VEL
LIN {X 0,Y 484.607,Z 784.208,A -85,B 0,C 180,E1 18858.725,E2 18858.725} C_VEL
LIN {X 0,Y 479.668,Z 809.429,A -85,B 0,C 180,E1 18857.643,E2 18857.643} C_VEL
LIN {X 0,Y 474.73,Z 830.911,A -85,B 0,C 180,E1 18856.516,E2 18856.516} C_VEL
LIN {X 0,Y 469.747,Z 850.543,A -85,B 0,C 180,E1 18855.311,E2 18855.311} C_VEL
LIN {X 0,Y 463.419,Z 873.405,A -85,B 0,C 180,E1 18853.665,E2 18853.665} C_VEL
LIN {X 0,Y 457.187,Z 893.771,A -85,B 0,C 180,E1 18851.923,E2 18851.923} C_VEL
LIN {X 0,Y 451.36,Z 911.899,A -85,B 0,C 180,E1 18850.139,E2 18850.139} C_VEL
LIN {X 0,Y 444.181,Z 933.171,A -85,B 0,C 180,E1 18847.69,E2 18847.69} C_VEL
LIN {X 0,Y 438.902,Z 948.239,A -85,B 0,C 180,E1 18845.676,E2 18845.676} C_VEL
LIN {X 0,Y 433.671,Z 963.005,A -85,B 0,C 180,E1 18843.439,E2 18843.439} C_VEL
LIN {X 0,Y 427.7,Z 979.892,A -85,B 0,C 180,E1 18840.484,E2 18840.484} C_VEL
LIN {X 0,Y 423.046,Z 993.229,A -85,B 0,C 180,E1 18837.75,E2 18837.75} C_VEL
LIN {X 0,Y 419.113,Z 1005.095,A -85,B 0,C 180,E1 18834.963,E2 18834.963} C_VEL
LIN {X 0,Y 415.071,Z 1018.205,A -85,B 0,C 180,E1 18831.331,E2 18831.331} C_VEL
LIN {X 0,Y 412.573,Z 1027.21,A -85,B 0,C 180,E1 18828.364,E2 18828.364} C_VEL
LIN {X 0,Y 410.593,Z 1035.625,A -85,B 0,C 180,E1 18825.104,E2 18825.104} C_VEL
LIN {X 0,Y 409.145,Z 1043.236,A -85,B 0,C 180,E1 18821.417,E2 18821.417} C_VEL
LIN {X 0,Y 408.452,Z 1048.085,A -85,B 0,C 180,E1 18818.446,E2 18818.446} C_VEL
LIN {X 0,Y 408.096,Z 1051.822,A -85,B 0,C 180,E1 18815.483,E2 18815.483} C_VEL
LIN {X 0,Y 407.945,Z 1054.407,A -85,B 0,C 180,E1 18812.611,E2 18812.611} C_VEL
LIN {X 0,Y 406.936,Z 1055.169,A -85,B 0,C 180,E1 18811.534,E2 18811.534} C_VEL
LIN {X 0,Y 400.45,Z 1056.363,A -85,B 0,C 180,E1 18808.49,E2 18808.49} C_VEL
LIN {X 0,Y 399.903,Z 1056.481,A -85,B 0,C 180,E1 18807.693,E2 18807.693} C_VEL
LIN {X 0,Y 399.922,Z 1056.217,A -85,B 0,C 180,E1 18804.26,E2 18804.26} C_VEL
LIN {X 0,Y 399.972,Z 1054.375,A -85,B 0,C 180,E1 18800.793,E2 18800.793} C_VEL
LIN {X 0,Y 400.149,Z 1051.786,A -85,B 0,C 180,E1 18797.884,E2 18797.884} C_VEL
LIN {X 0,Y 400.568,Z 1048.174,A -85,B 0,C 180,E1 18794.954,E2 18794.954} C_VEL
LIN {X 0,Y 401.392,Z 1043.256,A -85,B 0,C 180,E1 18791.858,E2 18791.858} C_VEL
LIN {X 0,Y 403.092,Z 1035.474,A -85,B 0,C 180,E1 18788.003,E2 18788.003} C_VEL
LIN {X 0,Y 405.308,Z 1027.265,A -85,B 0,C 180,E1 18784.736,E2 18784.736} C_VEL
LIN {X 0,Y 408.031,Z 1018.527,A -85,B 0,C 180,E1 18781.774,E2 18781.774} C_VEL
LIN {X 0,Y 412.48,Z 1005.687,A -85,B 0,C 180,E1 18778.099,E2 18778.099} C_VEL
LIN {X 0,Y 416.899,Z 993.667,A -85,B 0,C 180,E1 18775.193,E2 18775.193} C_VEL
LIN {X 0,Y 421.904,Z 980.764,A -85,B 0,C 180,E1 18772.477,E2 18772.477} C_VEL
LIN {X 0,Y 428.621,Z 963.608,A -85,B 0,C 180,E1 18769.394,E2 18769.394} C_VEL
LIN {X 0,Y 434.508,Z 948.519,A -85,B 0,C 180,E1 18767.066,E2 18767.066} C_VEL
LIN {X 0,Y 441.426,Z 930.638,A -85,B 0,C 180,E1 18764.663,E2 18764.663} C_VEL
LIN {X 0,Y 448.693,Z 910.831,A -85,B 0,C 180,E1 18762.413,E2 18762.413} C_VEL
LIN {X 0,Y 454.881,Z 893.213,A -85,B 0,C 180,E1 18760.681,E2 18760.681} C_VEL
LIN {X 0,Y 462.11,Z 871.436,A -85,B 0,C 180,E1 18758.836,E2 18758.836} C_VEL
LIN {X 0,Y 468.53,Z 849.906,A -85,B 0,C 180,E1 18757.307,E2 18757.307} C_VEL
LIN {X 0,Y 473.97,Z 830.063,A -85,B 0,C 180,E1 18756.101,E2 18756.101} C_VEL
LIN {X 0,Y 480.001,Z 805.386,A -85,B 0,C 180,E1 18754.841,E2 18754.841} C_VEL
LIN {X 0,Y 484.65,Z 782.962,A -85,B 0,C 180,E1 18753.913,E2 18753.913} C_VEL
LIN {X 0,Y 488.49,Z 761.416,A -85,B 0,C 180,E1 18753.184,E2 18753.184} C_VEL
LIN {X 0,Y 492.149,Z 736.286,A -85,B 0,C 180,E1 18752.513,E2 18752.513} C_VEL
LIN {X 0,Y 494.639,Z 711.25,A -85,B 0,C 180,E1 18752.019,E2 18752.019} C_VEL
LIN {X 0,Y 508.413,Z 484.25,A -85,B 0,C 180,E1 18748.469,E2 18748.469} C_VEL
LIN {X 0,Y 511.941,Z 426.076,A -85,B 0,C 180,E1 18747.543,E2 18747.543} C_VEL
LIN {X 0,Y 503.467,Z 412.199,A -85,B 0,C 180,E1 18745.34,E2 18745.34} C_VEL
LIN {X 0,Y 495.234,Z 400.273,A -85,B 0,C 180,E1 18742.997,E2 18742.997} C_VEL
LIN {X 0,Y 487.516,Z 389.775,A -85,B 0,C 180,E1 18740.531,E2 18740.531} C_VEL
LIN {X 0,Y 483.088,Z 384.047,A -85,B 0,C 180,E1 18738.963,E2 18738.963} C_VEL
LIN {X 0,Y 479.7,Z 379.554,A -85,B 0,C 180,E1 18737.655,E2 18737.655} C_VEL
LIN {X 0,Y 475.732,Z 374.454,A -85,B 0,C 180,E1 18735.982,E2 18735.982} C_VEL
LIN {X 0,Y 471.532,Z 369.115,A -85,B 0,C 180,E1 18733.989,E2 18733.989} C_VEL
LIN {X 0,Y 468.104,Z 365.104,A -85,B 0,C 180,E1 18732.146,E2 18732.146} C_VEL
LIN {X 0,Y 467.033,Z 363.453,A -85,B 0,C 180,E1 18731.485,E2 18731.485} C_VEL
LIN {X 0,Y 463.571,Z 359.825,A -85,B 0,C 180,E1 18729.184,E2 18729.184} C_VEL
LIN {X 0,Y 462.27,Z 357.505,A -85,B 0,C 180,E1 18728.082,E2 18728.082} C_VEL
LIN {X 0,Y 458.923,Z 354.474,A -85,B 0,C 180,E1 18724.749,E2 18724.749} C_VEL
LIN {X 0,Y 457.598,Z 351.664,A -85,B 0,C 180,E1 18722.379,E2 18722.379} C_VEL
LIN {X 0,Y 456.652,Z 351.021,A -85,B 0,C 180,E1 18718.369,E2 18718.369} C_VEL
LIN {X 0,Y 457.781,Z 351.809,A -85,B 0,C 180,E1 18714.359,E2 18714.359} C_VEL
LIN {X 0,Y 460.288,Z 356.205,A -85,B 0,C 180,E1 18710.749,E2 18710.749} C_VEL
LIN {X 0,Y 462.62,Z 357.915,A -85,B 0,C 180,E1 18708.72,E2 18708.72} C_VEL
LIN {X 0,Y 465.077,Z 361.723,A -85,B 0,C 180,E1 18706.827,E2 18706.827} C_VEL
LIN {X 0,Y 467.509,Z 364.088,A -85,B 0,C 180,E1 18705.319,E2 18705.319} C_VEL
LIN {X 0,Y 470.68,Z 368.369,A -85,B 0,C 180,E1 18703.525,E2 18703.525} C_VEL
LIN {X 0,Y 472.434,Z 370.226,A -85,B 0,C 180,E1 18702.654,E2 18702.654} C_VEL
LIN {X 0,Y 477.056,Z 376.185,A -85,B 0,C 180,E1 18700.533,E2 18700.533} C_VEL
LIN {X 0,Y 481.67,Z 382.188,A -85,B 0,C 180,E1 18698.666,E2 18698.666} C_VEL
LIN {X 0,Y 486.148,Z 388.097,A -85,B 0,C 180,E1 18697.029,E2 18697.029} C_VEL
LIN {X 0,Y 491.579,Z 396.101,A -85,B 0,C 180,E1 18695.196,E2 18695.196} C_VEL
LIN {X 0,Y 499.378,Z 407.801,A -85,B 0,C 180,E1 18692.837,E2 18692.837} C_VEL
LIN {X 0,Y 509.505,Z 424.348,A -85,B 0,C 180,E1 18690.101,E2 18690.101} C_VEL
LIN {X 0,Y 511.974,Z 428.804,A -85,B 0,C 180,E1 18689.474,E2 18689.474} C_VEL
LIN {X 0,Y 498.401,Z 651.761,A -85,B 0,C 180,E1 18685.999,E2 18685.999} C_VEL
LIN {X 0,Y 494.134,Z 720.659,A -85,B 0,C 180,E1 18684.902,E2 18684.902} C_VEL
LIN {X 0,Y 491.005,Z 748.417,A -85,B 0,C 180,E1 18684.318,E2 18684.318} C_VEL
LIN {X 0,Y 487.762,Z 769.54,A -85,B 0,C 180,E1 18683.739,E2 18683.739} C_VEL
LIN {X 0,Y 483.726,Z 791.614,A -85,B 0,C 180,E1 18682.982,E2 18682.982} C_VEL
LIN {X 0,Y 478.028,Z 817.744,A -85,B 0,C 180,E1 18681.857,E2 18681.857} C_VEL
LIN {X 0,Y 472.898,Z 838.162,A -85,B 0,C 180,E1 18680.787,E2 18680.787} C_VEL
LIN {X 0,Y 467.243,Z 858.592,A -85,B 0,C 180,E1 18679.531,E2 18679.531} C_VEL
LIN {X 0,Y 459.857,Z 882.625,A -85,B 0,C 180,E1 18677.772,E2 18677.772} C_VEL
LIN {X 0,Y 453.784,Z 900.866,A -85,B 0,C 180,E1 18676.198,E2 18676.198} C_VEL
LIN {X 0,Y 447.381,Z 919.119,A -85,B 0,C 180,E1 18674.391,E2 18674.391} C_VEL
LIN {X 0,Y 439.585,Z 940.175,A -85,B 0,C 180,E1 18671.943,E2 18671.943} C_VEL
LIN {X 0,Y 433.646,Z 955.71,A -85,B 0,C 180,E1 18669.841,E2 18669.841} C_VEL
LIN {X 0,Y 427.657,Z 971.27,A -85,B 0,C 180,E1 18667.437,E2 18667.437} C_VEL
LIN {X 0,Y 421.162,Z 988.077,A -85,B 0,C 180,E1 18664.405,E2 18664.405} C_VEL
LIN {X 0,Y 416.326,Z 1000.817,A -85,B 0,C 180,E1 18661.734,E2 18661.734} C_VEL
LIN {X 0,Y 411.664,Z 1013.865,A -85,B 0,C 180,E1 18658.587,E2 18658.587} C_VEL
LIN {X 0,Y 407.586,Z 1025.959,A -85,B 0,C 180,E1 18655.113,E2 18655.113} C_VEL
LIN {X 0,Y 404.988,Z 1034.645,A -85,B 0,C 180,E1 18652.194,E2 18652.194} C_VEL
LIN {X 0,Y 402.873,Z 1042.837,A -85,B 0,C 180,E1 18648.973,E2 18648.973} C_VEL
LIN {X 0,Y 401.25,Z 1050.659,A -85,B 0,C 180,E1 18645.168,E2 18645.168} C_VEL
LIN {X 0,Y 400.486,Z 1055.633,A -85,B 0,C 180,E1 18642.106,E2 18642.106} C_VEL
LIN {X 0,Y 400.097,Z 1059.326,A -85,B 0,C 180,E1 18639.193,E2 18639.193} C_VEL
LIN {X 0,Y 399.952,Z 1061.981,A -85,B 0,C 180,E1 18636.315,E2 18636.315} C_VEL
LIN {X 0,Y 399.914,Z 1063.923,A -85,B 0,C 180,E1 18632.866,E2 18632.866} C_VEL
LIN {X 0,Y 399.91,Z 1064.288,A -85,B 0,C 180,E1 18629.427,E2 18629.427} C_VEL
LIN {X 0,Y 399.912,Z 1063.465,A -85,B 0,C 180,E1 18626.416,E2 18626.416} C_VEL
LIN {X 0,Y 399.959,Z 1061.668,A -85,B 0,C 180,E1 18623.541,E2 18623.541} C_VEL
LIN {X 0,Y 400.109,Z 1058.86,A -85,B 0,C 180,E1 18620.652,E2 18620.652} C_VEL
LIN {X 0,Y 400.617,Z 1054.185,A -85,B 0,C 180,E1 18617.166,E2 18617.166} C_VEL
LIN {X 0,Y 401.678,Z 1047.5,A -85,B 0,C 180,E1 18613.514,E2 18613.514} C_VEL
LIN {X 0,Y 403.11,Z 1040.69,A -85,B 0,C 180,E1 18610.488,E2 18610.488} C_VEL
LIN {X 0,Y 405.362,Z 1031.948,A -85,B 0,C 180,E1 18607.216,E2 18607.216} C_VEL
LIN {X 0,Y 408.667,Z 1020.666,A -85,B 0,C 180,E1 18603.714,E2 18603.714} C_VEL
LIN {X 0,Y 412.193,Z 1009.732,A -85,B 0,C 180,E1 18600.818,E2 18600.818} C_VEL
LIN {X 0,Y 416.995,Z 996.039,A -85,B 0,C 180,E1 18597.675,E2 18597.675} C_VEL
LIN {X 0,Y 422.41,Z 980.801,A -85,B 0,C 180,E1 18594.72,E2 18594.72} C_VEL
LIN {X 0,Y 427.453,Z 966.939,A -85,B 0,C 180,E1 18592.373,E2 18592.373} C_VEL
LIN {X 0,Y 433.999,Z 949.133,A -85,B 0,C 180,E1 18589.741,E2 18589.741} C_VEL
LIN {X 0,Y 440.492,Z 930.708,A -85,B 0,C 180,E1 18587.434,E2 18587.434} C_VEL
